KUKA KRL data list: CNC6.dat

&ACCESS RV
DEFDAT CNC6 Public
DECL GLOBAL FRAME gfCNCPoint6[13477]


gfCNCPoint6[1] = {X 105.3781, Y 13.7586, Z -8.0000, A 0.000, B 0.000, C 0.000 }
gfCNCPoint6[2] = {X 105.3083, Y 12.9780, Z -8.0000, A 0.000, B 0.000, C 0.000 }
gfCNCPoint6[3] = {X 105.3083, Y 12.1868, Z -8.0000, A 0.000, B 0.000, C 0.000 }
gfCNCPoint6[4] = {X 105.4186, Y 11.2077, Z -8.0000, A 0.000, B 0.000, C 0.000 }
gfCNCPoint6[5] = {X 105.7440, Y 10.2777, Z -8.0000, A 0.000, B 0.000, C 0.000 }
gfCNCPoint6[6] = {X 106.2682, Y 9.4435, Z -8.0000, A 0.000, B 0.000, C 0.000 }
gfCNCPoint6[7] = {X 106.9649, Y 8.7468, Z -8.0000, A 0.000, B 0.000, C 0.000 }
gfCNCPoint6[8] = {X 107.7992, Y 8.2226, Z -8.0000, A 0.000, B 0.000, C 0.000 }
gfCNCPoint6[9] = {X 108.7292, Y 7.8971, Z -8.0000, A 0.000, B 0.000, C 0.000 }
gfCNCPoint6[10] = {X 109.7083, Y 7.7868, Z -8.0000, A 0.000, B 0.000, C 0.000 }
gfCNCPoint6[11] = {X 117.7916, Y 7.7868, Z -8.0000, A 0.000, B 0.000, C 0.000 }
gfCNCPoint6[12] = {X 118.7707, Y 7.8971, Z -8.0000, A 0.000, B 0.000, C 0.000 }
gfCNCPoint6[13] = {X 119.7007, Y 8.2226, Z -8.0000, A 0.000, B 0.000, C 0.000 }
gfCNCPoint6[14] = {X 120.5349, Y 8.7468, Z -8.0000, A 0.000, B 0.000, C 0.000 }
gfCNCPoint6[15] = {X 121.2316, Y 9.4435, Z -8.0000, A 0.000, B 0.000, C 0.000 }
gfCNCPoint6[16] = {X 121.7558, Y 10.2777, Z -8.0000, A 0.000, B 0.000, C 0.000 }
gfCNCPoint6[17] = {X 122.0813, Y 11.2077, Z -8.0000, A 0.000, B 0.000, C 0.000 }
gfCNCPoint6[18] = {X 122.1916, Y 12.1868, Z -8.0000, A 0.000, B 0.000, C 0.000 }
gfCNCPoint6[19] = {X 122.1913, Y 13.0233, Z -8.0000, A 0.000, B 0.000, C 0.000 }
gfCNCPoint6[20] = {X 122.0831, Y 13.9490, Z -8.0000, A 0.000, B 0.000, C 0.000 }
gfCNCPoint6[21] = {X 121.7823, Y 14.8311, Z -8.0000, A 0.000, B 0.000, C 0.000 }
gfCNCPoint6[22] = {X 121.3025, Y 15.6301, Z -8.0000, A 0.000, B 0.000, C 0.000 }
gfCNCPoint6[23] = {X 120.6651, Y 16.3101, Z -8.0000, A 0.000, B 0.000, C 0.000 }
gfCNCPoint6[24] = {X 120.6653, Y 40.8772, Z -8.0000, A 0.000, B 0.000, C 0.000 }
gfCNCPoint6[25] = {X 120.6784, Y 40.8882, Z -8.0000, A 0.000, B 0.000, C 0.000 }
gfCNCPoint6[26] = {X 121.3172, Y 41.5763, Z -8.0000, A 0.000, B 0.000, C 0.000 }
gfCNCPoint6[27] = {X 121.7955, Y 42.3843, Z -8.0000, A 0.000, B 0.000, C 0.000 }
gfCNCPoint6[28] = {X 122.0914, Y 43.2753, Z -8.0000, A 0.000, B 0.000, C 0.000 }
gfCNCPoint6[29] = {X 122.1916, Y 44.2089, Z -8.0000, A 0.000, B 0.000, C 0.000 }
gfCNCPoint6[30] = {X 122.1916, Y 45.0000, Z -8.0000, A 0.000, B 0.000, C 0.000 }
gfCNCPoint6[31] = {X 122.0813, Y 45.9791, Z -8.0000, A 0.000, B 0.000, C 0.000 }
gfCNCPoint6[32] = {X 121.7558, Y 46.9091, Z -8.0000, A 0.000, B 0.000, C 0.000 }
gfCNCPoint6[33] = {X 121.2316, Y 47.7434, Z -8.0000, A 0.000, B 0.000, C 0.000 }
gfCNCPoint6[34] = {X 120.5349, Y 48.4401, Z -8.0000, A 0.000, B 0.000, C 0.000 }
gfCNCPoint6[35] = {X 119.7007, Y 48.9643, Z -8.0000, A 0.000, B 0.000, C 0.000 }
gfCNCPoint6[36] = {X 118.7707, Y 49.2897, Z -8.0000, A 0.000, B 0.000, C 0.000 }
gfCNCPoint6[37] = {X 117.7916, Y 49.4000, Z -8.0000, A 0.000, B 0.000, C 0.000 }
gfCNCPoint6[38] = {X 111.9185, Y 49.4000, Z -8.0000, A 0.000, B 0.000, C 0.000 }
gfCNCPoint6[39] = {X 110.9394, Y 49.2897, Z -8.0000, A 0.000, B 0.000, C 0.000 }
gfCNCPoint6[40] = {X 110.0094, Y 48.9643, Z -8.0000, A 0.000, B 0.000, C 0.000 }
gfCNCPoint6[41] = {X 109.1751, Y 48.4401, Z -8.0000, A 0.000, B 0.000, C 0.000 }
gfCNCPoint6[42] = {X 108.4784, Y 47.7433, Z -8.0000, A 0.000, B 0.000, C 0.000 }
gfCNCPoint6[43] = {X 107.9542, Y 46.9091, Z -8.0000, A 0.000, B 0.000, C 0.000 }
gfCNCPoint6[44] = {X 107.6288, Y 45.9791, Z -8.0000, A 0.000, B 0.000, C 0.000 }
gfCNCPoint6[45] = {X 107.5185, Y 45.0000, Z -8.0000, A 0.000, B 0.000, C 0.000 }
gfCNCPoint6[46] = {X 107.5185, Y 44.1753, Z -8.0000, A 0.000, B 0.000, C 0.000 }
gfCNCPoint6[47] = {X 107.5542, Y 43.6267, Z -8.0000, A 0.000, B 0.000, C 0.000 }
gfCNCPoint6[48] = {X 107.6609, Y 43.0873, Z -8.0000, A 0.000, B 0.000, C 0.000 }
gfCNCPoint6[49] = {X 106.1856, Y 46.6923, Z -8.0000, A 0.000, B 0.000, C 0.000 }
gfCNCPoint6[50] = {X 105.8087, Y 47.4049, Z -8.0000, A 0.000, B 0.000, C 0.000 }
gfCNCPoint6[51] = {X 105.3081, Y 48.0367, Z -8.0000, A 0.000, B 0.000, C 0.000 }
gfCNCPoint6[52] = {X 104.7006, Y 48.5667, Z -8.0000, A 0.000, B 0.000, C 0.000 }
gfCNCPoint6[53] = {X 104.0067, Y 48.9769, Z -8.0000, A 0.000, B 0.000, C 0.000 }
gfCNCPoint6[54] = {X 103.0414, Y 49.3033, Z -8.0000, A 0.000, B 0.000, C 0.000 }
gfCNCPoint6[55] = {X 102.0269, Y 49.3989, Z -8.0000, A 0.000, B 0.000, C 0.000 }
gfCNCPoint6[56] = {X 101.0176, Y 49.2586, Z -8.0000, A 0.000, B 0.000, C 0.000 }
gfCNCPoint6[57] = {X 100.0676, Y 48.8899, Z -8.0000, A 0.000, B 0.000, C 0.000 }
gfCNCPoint6[58] = {X 99.2280, Y 48.3125, Z -8.0000, A 0.000, B 0.000, C 0.000 }
gfCNCPoint6[59] = {X 98.5436, Y 47.5575, Z -8.0000, A 0.000, B 0.000, C 0.000 }
gfCNCPoint6[60] = {X 98.0514, Y 46.6653, Z -8.0000, A 0.000, B 0.000, C 0.000 }
gfCNCPoint6[61] = {X 96.5899, Y 43.0909, Z -8.0000, A 0.000, B 0.000, C 0.000 }
gfCNCPoint6[62] = {X 96.6995, Y 43.6452, Z -8.0000, A 0.000, B 0.000, C 0.000 }
gfCNCPoint6[63] = {X 96.7385, Y 44.2088, Z -8.0000, A 0.000, B 0.000, C 0.000 }
gfCNCPoint6[64] = {X 96.7383, Y 45.0423, Z -8.0000, A 0.000, B 0.000, C 0.000 }
gfCNCPoint6[65] = {X 96.6200, Y 46.0144, Z -8.0000, A 0.000, B 0.000, C 0.000 }
gfCNCPoint6[66] = {X 96.2896, Y 46.9363, Z -8.0000, A 0.000, B 0.000, C 0.000 }
gfCNCPoint6[67] = {X 95.7635, Y 47.7622, Z -8.0000, A 0.000, B 0.000, C 0.000 }
gfCNCPoint6[68] = {X 95.0677, Y 48.4513, Z -8.0000, A 0.000, B 0.000, C 0.000 }
gfCNCPoint6[69] = {X 94.2367, Y 48.9695, Z -8.0000, A 0.000, B 0.000, C 0.000 }
gfCNCPoint6[70] = {X 93.3117, Y 49.2910, Z -8.0000, A 0.000, B 0.000, C 0.000 }
gfCNCPoint6[71] = {X 92.3385, Y 49.4000, Z -8.0000, A 0.000, B 0.000, C 0.000 }
gfCNCPoint6[72] = {X 85.8951, Y 49.4000, Z -8.0000, A 0.000, B 0.000, C 0.000 }
gfCNCPoint6[73] = {X 84.9160, Y 49.2897, Z -8.0000, A 0.000, B 0.000, C 0.000 }
gfCNCPoint6[74] = {X 83.9860, Y 48.9643, Z -8.0000, A 0.000, B 0.000, C 0.000 }
gfCNCPoint6[75] = {X 83.1517, Y 48.4401, Z -8.0000, A 0.000, B 0.000, C 0.000 }
gfCNCPoint6[76] = {X 82.4550, Y 47.7433, Z -8.0000, A 0.000, B 0.000, C 0.000 }
gfCNCPoint6[77] = {X 81.9308, Y 46.9091, Z -8.0000, A 0.000, B 0.000, C 0.000 }
gfCNCPoint6[78] = {X 81.6054, Y 45.9791, Z -8.0000, A 0.000, B 0.000, C 0.000 }
gfCNCPoint6[79] = {X 81.4951, Y 45.0000, Z -8.0000, A 0.000, B 0.000, C 0.000 }
gfCNCPoint6[80] = {X 81.4951, Y 44.2069, Z -8.0000, A 0.000, B 0.000, C 0.000 }
gfCNCPoint6[81] = {X 81.5995, Y 43.2694, Z -8.0000, A 0.000, B 0.000, C 0.000 }
gfCNCPoint6[82] = {X 81.8990, Y 42.3749, Z -8.0000, A 0.000, B 0.000, C 0.000 }
gfCNCPoint6[83] = {X 82.3802, Y 41.5636, Z -8.0000, A 0.000, B 0.000, C 0.000 }
gfCNCPoint6[84] = {X 83.0216, Y 40.8719, Z -8.0000, A 0.000, B 0.000, C 0.000 }
gfCNCPoint6[85] = {X 83.0217, Y 16.3102, Z -8.0000, A 0.000, B 0.000, C 0.000 }
gfCNCPoint6[86] = {X 82.3774, Y 15.6212, Z -8.0000, A 0.000, B 0.000, C 0.000 }
gfCNCPoint6[87] = {X 81.8949, Y 14.8106, Z -8.0000, A 0.000, B 0.000, C 0.000 }
gfCNCPoint6[88] = {X 81.5962, Y 13.9159, Z -8.0000, A 0.000, B 0.000, C 0.000 }
gfCNCPoint6[89] = {X 81.4951, Y 12.9780, Z -8.0000, A 0.000, B 0.000, C 0.000 }
gfCNCPoint6[90] = {X 81.4951, Y 12.1868, Z -8.0000, A 0.000, B 0.000, C 0.000 }
gfCNCPoint6[91] = {X 81.5776, Y 11.3387, Z -8.0000, A 0.000, B 0.000, C 0.000 }
gfCNCPoint6[92] = {X 81.8220, Y 10.5225, Z -8.0000, A 0.000, B 0.000, C 0.000 }
gfCNCPoint6[93] = {X 82.2192, Y 9.7686, Z -8.0000, A 0.000, B 0.000, C 0.000 }
gfCNCPoint6[94] = {X 81.8181, Y 9.5048, Z -8.0000, A 0.000, B 0.000, C 0.000 }
gfCNCPoint6[95] = {X 68.9232, Y 9.5048, Z -8.0000, A 0.000, B 0.000, C 0.000 }
gfCNCPoint6[96] = {X 69.1905, Y 10.7207, Z -8.0000, A 0.000, B 0.000, C 0.000 }
gfCNCPoint6[97] = {X 69.2995, Y 11.9609, Z -8.0000, A 0.000, B 0.000, C 0.000 }
gfCNCPoint6[98] = {X 69.3015, Y 12.0738, Z -8.0000, A 0.000, B 0.000, C 0.000 }
gfCNCPoint6[99] = {X 69.3021, Y 12.1868, Z -8.0000, A 0.000, B 0.000, C 0.000 }
gfCNCPoint6[100] = {X 69.3017, Y 13.0686, Z -8.0000, A 0.000, B 0.000, C 0.000 }
gfCNCPoint6[101] = {X 69.2128, Y 14.2897, Z -8.0000, A 0.000, B 0.000, C 0.000 }
gfCNCPoint6[102] = {X 68.9706, Y 15.4898, Z -8.0000, A 0.000, B 0.000, C 0.000 }
gfCNCPoint6[103] = {X 76.9202, Y 36.7547, Z -8.0000, A 0.000, B 0.000, C 0.000 }
gfCNCPoint6[104] = {X 77.6316, Y 37.4066, Z -8.0000, A 0.000, B 0.000, C 0.000 }
gfCNCPoint6[105] = {X 78.2746, Y 38.1261, Z -8.0000, A 0.000, B 0.000, C 0.000 }
gfCNCPoint6[106] = {X 79.0225, Y 39.1911, Z -8.0000, A 0.000, B 0.000, C 0.000 }
gfCNCPoint6[107] = {X 79.6207, Y 40.3468, Z -8.0000, A 0.000, B 0.000, C 0.000 }
gfCNCPoint6[108] = {X 80.0585, Y 41.5723, Z -8.0000, A 0.000, B 0.000, C 0.000 }
gfCNCPoint6[109] = {X 80.3280, Y 42.8454, Z -8.0000, A 0.000, B 0.000, C 0.000 }
gfCNCPoint6[110] = {X 80.4242, Y 44.1432, Z -8.0000, A 0.000, B 0.000, C 0.000 }
gfCNCPoint6[111] = {X 80.4245, Y 45.0000, Z -8.0000, A 0.000, B 0.000, C 0.000 }
gfCNCPoint6[112] = {X 80.3511, Y 46.1898, Z -8.0000, A 0.000, B 0.000, C 0.000 }
gfCNCPoint6[113] = {X 80.1320, Y 47.3615, Z -8.0000, A 0.000, B 0.000, C 0.000 }
gfCNCPoint6[114] = {X 79.7706, Y 48.4974, Z -8.0000, A 0.000, B 0.000, C 0.000 }
gfCNCPoint6[115] = {X 79.2722, Y 49.5803, Z -8.0000, A 0.000, B 0.000, C 0.000 }
gfCNCPoint6[116] = {X 78.4688, Y 50.8341, Z -8.0000, A 0.000, B 0.000, C 0.000 }
gfCNCPoint6[117] = {X 77.4826, Y 51.9498, Z -8.0000, A 0.000, B 0.000, C 0.000 }
gfCNCPoint6[118] = {X 76.3369, Y 52.9011, Z -8.0000, A 0.000, B 0.000, C 0.000 }
gfCNCPoint6[119] = {X 75.0589, Y 53.6653, Z -8.0000, A 0.000, B 0.000, C 0.000 }
gfCNCPoint6[120] = {X 73.6787, Y 54.2246, Z -8.0000, A 0.000, B 0.000, C 0.000 }
gfCNCPoint6[121] = {X 72.2292, Y 54.5655, Z -8.0000, A 0.000, B 0.000, C 0.000 }
gfCNCPoint6[122] = {X 70.7445, Y 54.6800, Z -8.0000, A 0.000, B 0.000, C 0.000 }
gfCNCPoint6[123] = {X 64.1851, Y 54.6800, Z -8.0000, A 0.000, B 0.000, C 0.000 }
gfCNCPoint6[124] = {X 62.7229, Y 54.5689, Z -8.0000, A 0.000, B 0.000, C 0.000 }
gfCNCPoint6[125] = {X 61.2943, Y 54.2383, Z -8.0000, A 0.000, B 0.000, C 0.000 }
gfCNCPoint6[126] = {X 59.9320, Y 53.6956, Z -8.0000, A 0.000, B 0.000, C 0.000 }
gfCNCPoint6[127] = {X 58.6673, Y 52.9534, Z -8.0000, A 0.000, B 0.000, C 0.000 }
gfCNCPoint6[128] = {X 57.5293, Y 52.0286, Z -8.0000, A 0.000, B 0.000, C 0.000 }
gfCNCPoint6[129] = {X 56.6337, Y 51.0563, Z -8.0000, A 0.000, B 0.000, C 0.000 }
gfCNCPoint6[130] = {X 55.8790, Y 49.9710, Z -8.0000, A 0.000, B 0.000, C 0.000 }
gfCNCPoint6[131] = {X 55.1243, Y 51.0563, Z -8.0000, A 0.000, B 0.000, C 0.000 }
gfCNCPoint6[132] = {X 54.2288, Y 52.0286, Z -8.0000, A 0.000, B 0.000, C 0.000 }
gfCNCPoint6[133] = {X 53.0907, Y 52.9534, Z -8.0000, A 0.000, B 0.000, C 0.000 }
gfCNCPoint6[134] = {X 51.8261, Y 53.6956, Z -8.0000, A 0.000, B 0.000, C 0.000 }
gfCNCPoint6[135] = {X 50.4638, Y 54.2383, Z -8.0000, A 0.000, B 0.000, C 0.000 }
gfCNCPoint6[136] = {X 49.0351, Y 54.5689, Z -8.0000, A 0.000, B 0.000, C 0.000 }
gfCNCPoint6[137] = {X 47.5729, Y 54.6800, Z -8.0000, A 0.000, B 0.000, C 0.000 }
gfCNCPoint6[138] = {X 40.6393, Y 54.6800, Z -8.0000, A 0.000, B 0.000, C 0.000 }
gfCNCPoint6[139] = {X 39.2448, Y 54.5790, Z -8.0000, A 0.000, B 0.000, C 0.000 }
gfCNCPoint6[140] = {X 37.8793, Y 54.2782, Z -8.0000, A 0.000, B 0.000, C 0.000 }
gfCNCPoint6[141] = {X 36.5715, Y 53.7838, Z -8.0000, A 0.000, B 0.000, C 0.000 }
gfCNCPoint6[142] = {X 35.3485, Y 53.1062, Z -8.0000, A 0.000, B 0.000, C 0.000 }
gfCNCPoint6[143] = {X 33.9151, Y 54.1351, Z -8.0000, A 0.000, B 0.000, C 0.000 }
gfCNCPoint6[144] = {X 32.3637, Y 54.9757, Z -8.0000, A 0.000, B 0.000, C 0.000 }
gfCNCPoint6[145] = {X 30.7189, Y 55.6147, Z -8.0000, A 0.000, B 0.000, C 0.000 }
gfCNCPoint6[146] = {X 29.0069, Y 56.0418, Z -8.0000, A 0.000, B 0.000, C 0.000 }
gfCNCPoint6[147] = {X 27.2548, Y 56.2503, Z -8.0000, A 0.000, B 0.000, C 0.000 }
gfCNCPoint6[148] = {X 24.9805, Y 57.2333, Z -8.0000, A 0.000, B 0.000, C 0.000 }
gfCNCPoint6[149] = {X 22.6486, Y 58.0704, Z -8.0000, A 0.000, B 0.000, C 0.000 }
gfCNCPoint6[150] = {X 20.0864, Y 58.7995, Z -8.0000, A 0.000, B 0.000, C 0.000 }
gfCNCPoint6[151] = {X 17.4731, Y 59.3158, Z -8.0000, A 0.000, B 0.000, C 0.000 }
gfCNCPoint6[152] = {X 14.8262, Y 59.6160, Z -8.0000, A 0.000, B 0.000, C 0.000 }
gfCNCPoint6[153] = {X 12.1636, Y 59.6979, Z -8.0000, A 0.000, B 0.000, C 0.000 }
gfCNCPoint6[154] = {X 9.5033, Y 59.5611, Z -8.0000, A 0.000, B 0.000, C 0.000 }
gfCNCPoint6[155] = {X 9.5033, Y 90.4952, Z -8.0000, A 0.000, B 0.000, C 0.000 }
gfCNCPoint6[156] = {X 114.8634, Y 90.4952, Z -8.0000, A 0.000, B 0.000, C 0.000 }
gfCNCPoint6[157] = {X 115.7474, Y 89.2996, Z -8.0000, A 0.000, B 0.000, C 0.000 }
gfCNCPoint6[158] = {X 116.7717, Y 88.2217, Z -8.0000, A 0.000, B 0.000, C 0.000 }
gfCNCPoint6[159] = {X 117.9206, Y 87.2778, Z -8.0000, A 0.000, B 0.000, C 0.000 }
gfCNCPoint6[160] = {X 119.1768, Y 86.4822, Z -8.0000, A 0.000, B 0.000, C 0.000 }
gfCNCPoint6[161] = {X 120.5212, Y 85.8469, Z -8.0000, A 0.000, B 0.000, C 0.000 }
gfCNCPoint6[162] = {X 121.9334, Y 85.3816, Z -8.0000, A 0.000, B 0.000, C 0.000 }
gfCNCPoint6[163] = {X 123.3922, Y 85.0934, Z -8.0000, A 0.000, B 0.000, C 0.000 }
gfCNCPoint6[164] = {X 123.5272, Y 84.9476, Z -8.0000, A 0.000, B 0.000, C 0.000 }
gfCNCPoint6[165] = {X 123.6609, Y 84.8006, Z -8.0000, A 0.000, B 0.000, C 0.000 }
gfCNCPoint6[166] = {X 147.2181, Y 58.9332, Z -8.0000, A 0.000, B 0.000, C 0.000 }
gfCNCPoint6[167] = {X 147.2180, Y 58.0000, Z -8.0000, A 0.000, B 0.000, C 0.000 }
gfCNCPoint6[168] = {X 147.2987, Y 56.6058, Z -8.0000, A 0.000, B 0.000, C 0.000 }
gfCNCPoint6[169] = {X 147.5398, Y 55.2303, Z -8.0000, A 0.000, B 0.000, C 0.000 }
gfCNCPoint6[170] = {X 148.0022, Y 53.7185, Z -8.0000, A 0.000, B 0.000, C 0.000 }
gfCNCPoint6[171] = {X 148.6580, Y 52.2800, Z -8.0000, A 0.000, B 0.000, C 0.000 }
gfCNCPoint6[172] = {X 143.0396, Y 52.2800, Z -8.0000, A 0.000, B 0.000, C 0.000 }
gfCNCPoint6[173] = {X 141.7807, Y 52.1703, Z -8.0000, A 0.000, B 0.000, C 0.000 }
gfCNCPoint6[174] = {X 140.5597, Y 51.8446, Z -8.0000, A 0.000, B 0.000, C 0.000 }
gfCNCPoint6[175] = {X 139.4134, Y 51.3126, Z -8.0000, A 0.000, B 0.000, C 0.000 }
gfCNCPoint6[176] = {X 138.3764, Y 50.5904, Z -8.0000, A 0.000, B 0.000, C 0.000 }
gfCNCPoint6[177] = {X 137.4799, Y 49.6998, Z -8.0000, A 0.000, B 0.000, C 0.000 }
gfCNCPoint6[178] = {X 136.7509, Y 48.6675, Z -8.0000, A 0.000, B 0.000, C 0.000 }
gfCNCPoint6[179] = {X 136.2114, Y 47.5248, Z -8.0000, A 0.000, B 0.000, C 0.000 }
gfCNCPoint6[180] = {X 135.8777, Y 46.3059, Z -8.0000, A 0.000, B 0.000, C 0.000 }
gfCNCPoint6[181] = {X 135.7598, Y 45.0477, Z -8.0000, A 0.000, B 0.000, C 0.000 }
gfCNCPoint6[182] = {X 135.7601, Y 44.1248, Z -8.0000, A 0.000, B 0.000, C 0.000 }
gfCNCPoint6[183] = {X 135.8408, Y 43.1249, Z -8.0000, A 0.000, B 0.000, C 0.000 }
gfCNCPoint6[184] = {X 136.0581, Y 42.1457, Z -8.0000, A 0.000, B 0.000, C 0.000 }
gfCNCPoint6[185] = {X 138.3597, Y 42.8258, Z -8.0000, A 0.000, B 0.000, C 0.000 }
gfCNCPoint6[186] = {X 138.6721, Y 42.0319, Z -8.0000, A 0.000, B 0.000, C 0.000 }
gfCNCPoint6[187] = {X 139.1179, Y 41.3046, Z -8.0000, A 0.000, B 0.000, C 0.000 }
gfCNCPoint6[188] = {X 139.6836, Y 40.6660, Z -8.0000, A 0.000, B 0.000, C 0.000 }
gfCNCPoint6[189] = {X 139.6836, Y 20.4384, Z -8.0000, A 0.000, B 0.000, C 0.000 }
gfCNCPoint6[190] = {X 137.7093, Y 20.4382, Z -8.0000, A 0.000, B 0.000, C 0.000 }
gfCNCPoint6[191] = {X 136.9994, Y 21.1828, Z -8.0000, A 0.000, B 0.000, C 0.000 }
gfCNCPoint6[192] = {X 136.1491, Y 21.7619, Z -8.0000, A 0.000, B 0.000, C 0.000 }
gfCNCPoint6[193] = {X 135.4282, Y 22.0767, Z -8.0000, A 0.000, B 0.000, C 0.000 }
gfCNCPoint6[194] = {X 134.6660, Y 22.2715, Z -8.0000, A 0.000, B 0.000, C 0.000 }
gfCNCPoint6[195] = {X 133.8824, Y 22.3414, Z -8.0000, A 0.000, B 0.000, C 0.000 }
gfCNCPoint6[196] = {X 133.2006, Y 22.3415, Z -8.0000, A 0.000, B 0.000, C 0.000 }
gfCNCPoint6[197] = {X 132.2486, Y 22.2478, Z -8.0000, A 0.000, B 0.000, C 0.000 }
gfCNCPoint6[198] = {X 131.3331, Y 21.9701, Z -8.0000, A 0.000, B 0.000, C 0.000 }
gfCNCPoint6[199] = {X 130.4895, Y 21.5191, Z -8.0000, A 0.000, B 0.000, C 0.000 }
gfCNCPoint6[200] = {X 129.7500, Y 20.9122, Z -8.0000, A 0.000, B 0.000, C 0.000 }
gfCNCPoint6[201] = {X 129.1431, Y 20.1727, Z -8.0000, A 0.000, B 0.000, C 0.000 }
gfCNCPoint6[202] = {X 128.6921, Y 19.3290, Z -8.0000, A 0.000, B 0.000, C 0.000 }
gfCNCPoint6[203] = {X 128.4144, Y 18.4136, Z -8.0000, A 0.000, B 0.000, C 0.000 }
gfCNCPoint6[204] = {X 128.3206, Y 17.4615, Z -8.0000, A 0.000, B 0.000, C 0.000 }
gfCNCPoint6[205] = {X 128.3206, Y 10.4835, Z -8.0000, A 0.000, B 0.000, C 0.000 }
gfCNCPoint6[206] = {X 128.3317, Y 10.1547, Z -8.0000, A 0.000, B 0.000, C 0.000 }
gfCNCPoint6[207] = {X 128.3649, Y 9.8275, Z -8.0000, A 0.000, B 0.000, C 0.000 }
gfCNCPoint6[208] = {X 128.6079, Y 8.8340, Z -8.0000, A 0.000, B 0.000, C 0.000 }
gfCNCPoint6[209] = {X 129.0526, Y 7.9130, Z -8.0000, A 0.000, B 0.000, C 0.000 }
gfCNCPoint6[210] = {X 129.6794, Y 7.1048, Z -8.0000, A 0.000, B 0.000, C 0.000 }
gfCNCPoint6[211] = {X 130.0258, Y 7.4372, Z -8.0000, A 0.000, B 0.000, C 0.000 }
gfCNCPoint6[212] = {X 130.6998, Y 6.8633, Z -8.0000, A 0.000, B 0.000, C 0.000 }
gfCNCPoint6[213] = {X 131.4750, Y 6.4360, Z -8.0000, A 0.000, B 0.000, C 0.000 }
gfCNCPoint6[214] = {X 132.3200, Y 6.1725, Z -8.0000, A 0.000, B 0.000, C 0.000 }
gfCNCPoint6[215] = {X 133.2007, Y 6.0835, Z -8.0000, A 0.000, B 0.000, C 0.000 }
gfCNCPoint6[216] = {X 133.8874, Y 6.0837, Z -8.0000, A 0.000, B 0.000, C 0.000 }
gfCNCPoint6[217] = {X 134.7185, Y 6.1716, Z -8.0000, A 0.000, B 0.000, C 0.000 }
gfCNCPoint6[218] = {X 135.5180, Y 6.4151, Z -8.0000, A 0.000, B 0.000, C 0.000 }
gfCNCPoint6[219] = {X 136.2570, Y 6.8053, Z -8.0000, A 0.000, B 0.000, C 0.000 }
gfCNCPoint6[220] = {X 136.9090, Y 7.3283, Z -8.0000, A 0.000, B 0.000, C 0.000 }
gfCNCPoint6[221] = {X 137.4502, Y 7.9650, Z -8.0000, A 0.000, B 0.000, C 0.000 }
gfCNCPoint6[222] = {X 155.0725, Y 7.9650, Z -8.0000, A 0.000, B 0.000, C 0.000 }
gfCNCPoint6[223] = {X 155.6203, Y 7.3220, Z -8.0000, A 0.000, B 0.000, C 0.000 }
gfCNCPoint6[224] = {X 156.2808, Y 6.7954, Z -8.0000, A 0.000, B 0.000, C 0.000 }
gfCNCPoint6[225] = {X 157.0298, Y 6.4048, Z -8.0000, A 0.000, B 0.000, C 0.000 }
gfCNCPoint6[226] = {X 157.8397, Y 6.1646, Z -8.0000, A 0.000, B 0.000, C 0.000 }
gfCNCPoint6[227] = {X 158.6805, Y 6.0835, Z -8.0000, A 0.000, B 0.000, C 0.000 }
gfCNCPoint6[228] = {X 159.3791, Y 6.0839, Z -8.0000, A 0.000, B 0.000, C 0.000 }
gfCNCPoint6[229] = {X 160.3488, Y 6.2050, Z -8.0000, A 0.000, B 0.000, C 0.000 }
gfCNCPoint6[230] = {X 161.2678, Y 6.5371, Z -8.0000, A 0.000, B 0.000, C 0.000 }
gfCNCPoint6[231] = {X 162.0908, Y 7.0639, Z -8.0000, A 0.000, B 0.000, C 0.000 }
gfCNCPoint6[232] = {X 162.7773, Y 7.7593, Z -8.0000, A 0.000, B 0.000, C 0.000 }
gfCNCPoint6[233] = {X 163.2934, Y 8.5891, Z -8.0000, A 0.000, B 0.000, C 0.000 }
gfCNCPoint6[234] = {X 163.6136, Y 9.5124, Z -8.0000, A 0.000, B 0.000, C 0.000 }
gfCNCPoint6[235] = {X 163.7221, Y 10.4835, Z -8.0000, A 0.000, B 0.000, C 0.000 }
gfCNCPoint6[236] = {X 163.7221, Y 17.4615, Z -8.0000, A 0.000, B 0.000, C 0.000 }
gfCNCPoint6[237] = {X 163.6118, Y 18.4406, Z -8.0000, A 0.000, B 0.000, C 0.000 }
gfCNCPoint6[238] = {X 163.2863, Y 19.3706, Z -8.0000, A 0.000, B 0.000, C 0.000 }
gfCNCPoint6[239] = {X 162.7621, Y 20.2049, Z -8.0000, A 0.000, B 0.000, C 0.000 }
gfCNCPoint6[240] = {X 162.0654, Y 20.9016, Z -8.0000, A 0.000, B 0.000, C 0.000 }
gfCNCPoint6[241] = {X 161.2312, Y 21.4258, Z -8.0000, A 0.000, B 0.000, C 0.000 }
gfCNCPoint6[242] = {X 160.3012, Y 21.7512, Z -8.0000, A 0.000, B 0.000, C 0.000 }
gfCNCPoint6[243] = {X 159.3221, Y 21.8615, Z -8.0000, A 0.000, B 0.000, C 0.000 }
gfCNCPoint6[244] = {X 158.6792, Y 21.8615, Z -8.0000, A 0.000, B 0.000, C 0.000 }
gfCNCPoint6[245] = {X 157.8337, Y 21.7773, Z -8.0000, A 0.000, B 0.000, C 0.000 }
gfCNCPoint6[246] = {X 157.0198, Y 21.5332, Z -8.0000, A 0.000, B 0.000, C 0.000 }
gfCNCPoint6[247] = {X 156.2675, Y 21.1381, Z -8.0000, A 0.000, B 0.000, C 0.000 }
gfCNCPoint6[248] = {X 155.6045, Y 20.6066, Z -8.0000, A 0.000, B 0.000, C 0.000 }
gfCNCPoint6[249] = {X 155.0552, Y 19.9583, Z -8.0000, A 0.000, B 0.000, C 0.000 }
gfCNCPoint6[250] = {X 152.3574, Y 19.9591, Z -8.0000, A 0.000, B 0.000, C 0.000 }
gfCNCPoint6[251] = {X 152.3564, Y 40.8428, Z -8.0000, A 0.000, B 0.000, C 0.000 }
gfCNCPoint6[252] = {X 152.8071, Y 41.3287, Z -8.0000, A 0.000, B 0.000, C 0.000 }
gfCNCPoint6[253] = {X 152.9013, Y 41.4409, Z -8.0000, A 0.000, B 0.000, C 0.000 }
gfCNCPoint6[254] = {X 153.4357, Y 42.2811, Z -8.0000, A 0.000, B 0.000, C 0.000 }
gfCNCPoint6[255] = {X 153.7686, Y 43.2196, Z -8.0000, A 0.000, B 0.000, C 0.000 }
gfCNCPoint6[256] = {X 153.8831, Y 44.2088, Z -8.0000, A 0.000, B 0.000, C 0.000 }
gfCNCPoint6[257] = {X 153.8829, Y 45.0423, Z -8.0000, A 0.000, B 0.000, C 0.000 }
gfCNCPoint6[258] = {X 153.7646, Y 46.0144, Z -8.0000, A 0.000, B 0.000, C 0.000 }
gfCNCPoint6[259] = {X 153.4342, Y 46.9363, Z -8.0000, A 0.000, B 0.000, C 0.000 }
gfCNCPoint6[260] = {X 152.9080, Y 47.7622, Z -8.0000, A 0.000, B 0.000, C 0.000 }
gfCNCPoint6[261] = {X 152.2123, Y 48.4513, Z -8.0000, A 0.000, B 0.000, C 0.000 }
gfCNCPoint6[262] = {X 151.3813, Y 48.9695, Z -8.0000, A 0.000, B 0.000, C 0.000 }
gfCNCPoint6[263] = {X 150.4563, Y 49.2910, Z -8.0000, A 0.000, B 0.000, C 0.000 }
gfCNCPoint6[264] = {X 149.4831, Y 49.4000, Z -8.0000, A 0.000, B 0.000, C 0.000 }
gfCNCPoint6[265] = {X 143.0396, Y 49.4000, Z -8.0000, A 0.000, B 0.000, C 0.000 }
gfCNCPoint6[266] = {X 142.0605, Y 49.2897, Z -8.0000, A 0.000, B 0.000, C 0.000 }
gfCNCPoint6[267] = {X 141.1305, Y 48.9643, Z -8.0000, A 0.000, B 0.000, C 0.000 }
gfCNCPoint6[268] = {X 140.2963, Y 48.4401, Z -8.0000, A 0.000, B 0.000, C 0.000 }
gfCNCPoint6[269] = {X 139.5996, Y 47.7433, Z -8.0000, A 0.000, B 0.000, C 0.000 }
gfCNCPoint6[270] = {X 139.0754, Y 46.9091, Z -8.0000, A 0.000, B 0.000, C 0.000 }
gfCNCPoint6[271] = {X 138.7499, Y 45.9791, Z -8.0000, A 0.000, B 0.000, C 0.000 }
gfCNCPoint6[272] = {X 138.6396, Y 45.0000, Z -8.0000, A 0.000, B 0.000, C 0.000 }
gfCNCPoint6[273] = {X 138.6400, Y 44.1483, Z -8.0000, A 0.000, B 0.000, C 0.000 }
gfCNCPoint6[274] = {X 138.7505, Y 43.2275, Z -8.0000, A 0.000, B 0.000, C 0.000 }
gfCNCPoint6[275] = {X 139.0514, Y 42.3503, Z -8.0000, A 0.000, B 0.000, C 0.000 }
gfCNCPoint6[276] = {X 139.5295, Y 41.5556, Z -8.0000, A 0.000, B 0.000, C 0.000 }
gfCNCPoint6[277] = {X 140.1636, Y 40.8789, Z -8.0000, A 0.000, B 0.000, C 0.000 }
gfCNCPoint6[278] = {X 140.1636, Y 19.9585, Z -8.0000, A 0.000, B 0.000, C 0.000 }
gfCNCPoint6[279] = {X 137.4654, Y 19.9582, Z -8.0000, A 0.000, B 0.000, C 0.000 }
gfCNCPoint6[280] = {X 136.9177, Y 20.6083, Z -8.0000, A 0.000, B 0.000, C 0.000 }
gfCNCPoint6[281] = {X 136.2552, Y 21.1409, Z -8.0000, A 0.000, B 0.000, C 0.000 }
gfCNCPoint6[282] = {X 135.5027, Y 21.5362, Z -8.0000, A 0.000, B 0.000, C 0.000 }
gfCNCPoint6[283] = {X 134.6883, Y 21.7794, Z -8.0000, A 0.000, B 0.000, C 0.000 }
gfCNCPoint6[284] = {X 133.8422, Y 21.8615, Z -8.0000, A 0.000, B 0.000, C 0.000 }
gfCNCPoint6[285] = {X 133.2006, Y 21.8615, Z -8.0000, A 0.000, B 0.000, C 0.000 }
gfCNCPoint6[286] = {X 132.2215, Y 21.7512, Z -8.0000, A 0.000, B 0.000, C 0.000 }
gfCNCPoint6[287] = {X 131.2916, Y 21.4258, Z -8.0000, A 0.000, B 0.000, C 0.000 }
gfCNCPoint6[288] = {X 130.4573, Y 20.9016, Z -8.0000, A 0.000, B 0.000, C 0.000 }
gfCNCPoint6[289] = {X 129.7606, Y 20.2049, Z -8.0000, A 0.000, B 0.000, C 0.000 }
gfCNCPoint6[290] = {X 129.2364, Y 19.3706, Z -8.0000, A 0.000, B 0.000, C 0.000 }
gfCNCPoint6[291] = {X 128.9110, Y 18.4406, Z -8.0000, A 0.000, B 0.000, C 0.000 }
gfCNCPoint6[292] = {X 128.8006, Y 17.4615, Z -8.0000, A 0.000, B 0.000, C 0.000 }
gfCNCPoint6[293] = {X 128.8006, Y 10.4835, Z -8.0000, A 0.000, B 0.000, C 0.000 }
gfCNCPoint6[294] = {X 128.8808, Y 9.6474, Z -8.0000, A 0.000, B 0.000, C 0.000 }
gfCNCPoint6[295] = {X 129.1184, Y 8.8418, Z -8.0000, A 0.000, B 0.000, C 0.000 }
gfCNCPoint6[296] = {X 129.5048, Y 8.0960, Z -8.0000, A 0.000, B 0.000, C 0.000 }
gfCNCPoint6[297] = {X 130.0258, Y 7.4372, Z -8.0000, A 0.000, B 0.000, C 0.000 }
gfCNCPoint6[298] = {X 129.6794, Y 7.1048, Z -8.0000, A 0.000, B 0.000, C 0.000 }
gfCNCPoint6[299] = {X 102.4337, Y 7.1048, Z -8.0000, A 0.000, B 0.000, C 0.000 }
gfCNCPoint6[300] = {X 102.4337, Y 11.9048, Z -8.0000, A 0.000, B 0.000, C 0.000 }
gfCNCPoint6[301] = {X 101.3242, Y 11.9048, Z -8.0000, A 0.000, B 0.000, C 0.000 }
gfCNCPoint6[302] = {X 101.3283, Y 12.0458, Z -8.0000, A 0.000, B 0.000, C 0.000 }
gfCNCPoint6[303] = {X 101.3297, Y 12.1868, Z -8.0000, A 0.000, B 0.000, C 0.000 }
gfCNCPoint6[304] = {X 101.3293, Y 13.0462, Z -8.0000, A 0.000, B 0.000, C 0.000 }
gfCNCPoint6[305] = {X 101.2276, Y 14.1928, Z -8.0000, A 0.000, B 0.000, C 0.000 }
gfCNCPoint6[306] = {X 100.9464, Y 15.3090, Z -8.0000, A 0.000, B 0.000, C 0.000 }
gfCNCPoint6[307] = {X 101.3187, Y 16.2359, Z -8.0000, A 0.000, B 0.000, C 0.000 }
gfCNCPoint6[308] = {X 101.8679, Y 17.5961, Z -8.0000, A 0.000, B 0.000, C 0.000 }
gfCNCPoint6[309] = {X 102.6897, Y 15.5479, Z -8.0000, A 0.000, B 0.000, C 0.000 }
gfCNCPoint6[310] = {X 102.7997, Y 15.2735, Z -8.0000, A 0.000, B 0.000, C 0.000 }
gfCNCPoint6[311] = {X 102.5272, Y 14.1739, Z -8.0000, A 0.000, B 0.000, C 0.000 }
gfCNCPoint6[312] = {X 102.4286, Y 13.0454, Z -8.0000, A 0.000, B 0.000, C 0.000 }
gfCNCPoint6[313] = {X 102.4283, Y 12.1868, Z -8.0000, A 0.000, B 0.000, C 0.000 }
gfCNCPoint6[314] = {X 102.4296, Y 12.0458, Z -8.0000, A 0.000, B 0.000, C 0.000 }
gfCNCPoint6[315] = {X 102.4337, Y 11.9048, Z -8.0000, A 0.000, B 0.000, C 0.000 }
gfCNCPoint6[316] = {X 102.4337, Y 9.5048, Z -8.0000, A 0.000, B 0.000, C 0.000 }
gfCNCPoint6[317] = {X 98.1266, Y 9.5048, Z -8.0000, A 0.000, B 0.000, C 0.000 }
gfCNCPoint6[318] = {X 98.5429, Y 10.2827, Z -8.0000, A 0.000, B 0.000, C 0.000 }
gfCNCPoint6[319] = {X 98.8123, Y 11.1229, Z -8.0000, A 0.000, B 0.000, C 0.000 }
gfCNCPoint6[320] = {X 98.9260, Y 11.9978, Z -8.0000, A 0.000, B 0.000, C 0.000 }
gfCNCPoint6[321] = {X 98.9288, Y 12.0923, Z -8.0000, A 0.000, B 0.000, C 0.000 }
gfCNCPoint6[322] = {X 98.9297, Y 12.1868, Z -8.0000, A 0.000, B 0.000, C 0.000 }
gfCNCPoint6[323] = {X 98.9294, Y 13.0237, Z -8.0000, A 0.000, B 0.000, C 0.000 }
gfCNCPoint6[324] = {X 98.8590, Y 13.8052, Z -8.0000, A 0.000, B 0.000, C 0.000 }
gfCNCPoint6[325] = {X 98.6643, Y 14.5654, Z -8.0000, A 0.000, B 0.000, C 0.000 }
gfCNCPoint6[326] = {X 98.3502, Y 15.2845, Z -8.0000, A 0.000, B 0.000, C 0.000 }
gfCNCPoint6[327] = {X 99.0924, Y 17.1324, Z -8.0000, A 0.000, B 0.000, C 0.000 }
gfCNCPoint6[328] = {X 101.8751, Y 24.0238, Z -8.0000, A 0.000, B 0.000, C 0.000 }
gfCNCPoint6[329] = {X 104.9172, Y 16.4412, Z -8.0000, A 0.000, B 0.000, C 0.000 }
gfCNCPoint6[330] = {X 105.3924, Y 15.2557, Z -8.0000, A 0.000, B 0.000, C 0.000 }
gfCNCPoint6[331] = {X 105.0866, Y 14.5446, Z -8.0000, A 0.000, B 0.000, C 0.000 }
gfCNCPoint6[332] = {X 104.8970, Y 13.7941, Z -8.0000, A 0.000, B 0.000, C 0.000 }
gfCNCPoint6[333] = {X 104.8285, Y 13.0231, Z -8.0000, A 0.000, B 0.000, C 0.000 }
gfCNCPoint6[334] = {X 104.8283, Y 12.1868, Z -8.0000, A 0.000, B 0.000, C 0.000 }
gfCNCPoint6[335] = {X 104.8292, Y 12.0923, Z -8.0000, A 0.000, B 0.000, C 0.000 }
gfCNCPoint6[336] = {X 104.8319, Y 11.9978, Z -8.0000, A 0.000, B 0.000, C 0.000 }
gfCNCPoint6[337] = {X 104.9457, Y 11.1229, Z -8.0000, A 0.000, B 0.000, C 0.000 }
gfCNCPoint6[338] = {X 105.2151, Y 10.2827, Z -8.0000, A 0.000, B 0.000, C 0.000 }
gfCNCPoint6[339] = {X 105.6313, Y 9.5048, Z -8.0000, A 0.000, B 0.000, C 0.000 }
gfCNCPoint6[340] = {X 102.4337, Y 9.5048, Z -8.0000, A 0.000, B 0.000, C 0.000 }
gfCNCPoint6[341] = {X 102.4337, Y 7.1048, Z -8.0000, A 0.000, B 0.000, C 0.000 }
gfCNCPoint6[342] = {X 64.8348, Y 7.1048, Z -8.0000, A 0.000, B 0.000, C 0.000 }
gfCNCPoint6[343] = {X 65.5945, Y 8.0240, Z -8.0000, A 0.000, B 0.000, C 0.000 }
gfCNCPoint6[344] = {X 66.1940, Y 9.0549, Z -8.0000, A 0.000, B 0.000, C 0.000 }
gfCNCPoint6[345] = {X 66.6171, Y 10.1698, Z -8.0000, A 0.000, B 0.000, C 0.000 }
gfCNCPoint6[346] = {X 66.8305, Y 11.1683, Z -8.0000, A 0.000, B 0.000, C 0.000 }
gfCNCPoint6[347] = {X 66.9021, Y 12.1868, Z -8.0000, A 0.000, B 0.000, C 0.000 }
gfCNCPoint6[348] = {X 66.9018, Y 13.0462, Z -8.0000, A 0.000, B 0.000, C 0.000 }
gfCNCPoint6[349] = {X 66.7774, Y 14.3201, Z -8.0000, A 0.000, B 0.000, C 0.000 }
gfCNCPoint6[350] = {X 66.4317, Y 15.5524, Z -8.0000, A 0.000, B 0.000, C 0.000 }
gfCNCPoint6[351] = {X 74.9135, Y 38.2407, Z -8.0000, A 0.000, B 0.000, C 0.000 }
gfCNCPoint6[352] = {X 75.8052, Y 38.9755, Z -8.0000, A 0.000, B 0.000, C 0.000 }
gfCNCPoint6[353] = {X 76.5695, Y 39.8422, Z -8.0000, A 0.000, B 0.000, C 0.000 }
gfCNCPoint6[354] = {X 77.1870, Y 40.8188, Z -8.0000, A 0.000, B 0.000, C 0.000 }
gfCNCPoint6[355] = {X 77.6422, Y 41.8809, Z -8.0000, A 0.000, B 0.000, C 0.000 }
gfCNCPoint6[356] = {X 77.9237, Y 43.0016, Z -8.0000, A 0.000, B 0.000, C 0.000 }
gfCNCPoint6[357] = {X 78.0243, Y 44.1527, Z -8.0000, A 0.000, B 0.000, C 0.000 }
gfCNCPoint6[358] = {X 78.0245, Y 45.0000, Z -8.0000, A 0.000, B 0.000, C 0.000 }
gfCNCPoint6[359] = {X 77.9139, Y 46.2642, Z -8.0000, A 0.000, B 0.000, C 0.000 }
gfCNCPoint6[360] = {X 77.5854, Y 47.4899, Z -8.0000, A 0.000, B 0.000, C 0.000 }
gfCNCPoint6[361] = {X 77.0491, Y 48.6400, Z -8.0000, A 0.000, B 0.000, C 0.000 }
gfCNCPoint6[362] = {X 76.3213, Y 49.6795, Z -8.0000, A 0.000, B 0.000, C 0.000 }
gfCNCPoint6[363] = {X 75.4240, Y 50.5768, Z -8.0000, A 0.000, B 0.000, C 0.000 }
gfCNCPoint6[364] = {X 74.3845, Y 51.3047, Z -8.0000, A 0.000, B 0.000, C 0.000 }
gfCNCPoint6[365] = {X 73.2344, Y 51.8410, Z -8.0000, A 0.000, B 0.000, C 0.000 }
gfCNCPoint6[366] = {X 72.0086, Y 52.1694, Z -8.0000, A 0.000, B 0.000, C 0.000 }
gfCNCPoint6[367] = {X 70.7445, Y 52.2800, Z -8.0000, A 0.000, B 0.000, C 0.000 }
gfCNCPoint6[368] = {X 64.1851, Y 52.2800, Z -8.0000, A 0.000, B 0.000, C 0.000 }
gfCNCPoint6[369] = {X 62.9397, Y 52.1727, Z -8.0000, A 0.000, B 0.000, C 0.000 }
gfCNCPoint6[370] = {X 61.7311, Y 51.8539, Z -8.0000, A 0.000, B 0.000, C 0.000 }
gfCNCPoint6[371] = {X 60.5947, Y 51.3330, Z -8.0000, A 0.000, B 0.000, C 0.000 }
gfCNCPoint6[372] = {X 59.5643, Y 50.6255, Z -8.0000, A 0.000, B 0.000, C 0.000 }
gfCNCPoint6[373] = {X 58.6700, Y 49.7521, Z -8.0000, A 0.000, B 0.000, C 0.000 }
gfCNCPoint6[374] = {X 57.9384, Y 48.7385, Z -8.0000, A 0.000, B 0.000, C 0.000 }
gfCNCPoint6[375] = {X 57.3706, Y 47.5614, Z -8.0000, A 0.000, B 0.000, C 0.000 }
gfCNCPoint6[376] = {X 57.0224, Y 46.3017, Z -8.0000, A 0.000, B 0.000, C 0.000 }
gfCNCPoint6[377] = {X 56.9051, Y 45.0000, Z -8.0000, A 0.000, B 0.000, C 0.000 }
gfCNCPoint6[378] = {X 56.9052, Y 44.1968, Z -8.0000, A 0.000, B 0.000, C 0.000 }
gfCNCPoint6[379] = {X 56.9289, Y 43.6212, Z -8.0000, A 0.000, B 0.000, C 0.000 }
gfCNCPoint6[380] = {X 56.9981, Y 43.0492, Z -8.0000, A 0.000, B 0.000, C 0.000 }
gfCNCPoint6[381] = {X 54.7600, Y 43.0492, Z -8.0000, A 0.000, B 0.000, C 0.000 }
gfCNCPoint6[382] = {X 54.8275, Y 43.6012, Z -8.0000, A 0.000, B 0.000, C 0.000 }
gfCNCPoint6[383] = {X 54.8528, Y 44.1567, Z -8.0000, A 0.000, B 0.000, C 0.000 }
gfCNCPoint6[384] = {X 54.8529, Y 45.0000, Z -8.0000, A 0.000, B 0.000, C 0.000 }
gfCNCPoint6[385] = {X 54.7356, Y 46.3017, Z -8.0000, A 0.000, B 0.000, C 0.000 }
gfCNCPoint6[386] = {X 54.3875, Y 47.5614, Z -8.0000, A 0.000, B 0.000, C 0.000 }
gfCNCPoint6[387] = {X 53.8197, Y 48.7385, Z -8.0000, A 0.000, B 0.000, C 0.000 }
gfCNCPoint6[388] = {X 53.0880, Y 49.7521, Z -8.0000, A 0.000, B 0.000, C 0.000 }
gfCNCPoint6[389] = {X 52.1938, Y 50.6255, Z -8.0000, A 0.000, B 0.000, C 0.000 }
gfCNCPoint6[390] = {X 51.1633, Y 51.3330, Z -8.0000, A 0.000, B 0.000, C 0.000 }
gfCNCPoint6[391] = {X 50.0270, Y 51.8539, Z -8.0000, A 0.000, B 0.000, C 0.000 }
gfCNCPoint6[392] = {X 48.8183, Y 52.1727, Z -8.0000, A 0.000, B 0.000, C 0.000 }
gfCNCPoint6[393] = {X 47.5729, Y 52.2800, Z -8.0000, A 0.000, B 0.000, C 0.000 }
gfCNCPoint6[394] = {X 40.6393, Y 52.2800, Z -8.0000, A 0.000, B 0.000, C 0.000 }
gfCNCPoint6[395] = {X 39.4476, Y 52.1818, Z -8.0000, A 0.000, B 0.000, C 0.000 }
gfCNCPoint6[396] = {X 38.2881, Y 51.8899, Z -8.0000, A 0.000, B 0.000, C 0.000 }
gfCNCPoint6[397] = {X 37.1919, Y 51.4120, Z -8.0000, A 0.000, B 0.000, C 0.000 }
gfCNCPoint6[398] = {X 36.1888, Y 50.7612, Z -8.0000, A 0.000, B 0.000, C 0.000 }
gfCNCPoint6[399] = {X 35.3058, Y 49.9550, Z -8.0000, A 0.000, B 0.000, C 0.000 }
gfCNCPoint6[400] = {X 34.8234, Y 50.4196, Z -8.0000, A 0.000, B 0.000, C 0.000 }
gfCNCPoint6[401] = {X 34.3150, Y 50.8555, Z -8.0000, A 0.000, B 0.000, C 0.000 }
gfCNCPoint6[402] = {X 33.7814, Y 51.2869, Z -8.0000, A 0.000, B 0.000, C 0.000 }
gfCNCPoint6[403] = {X 32.5222, Y 52.1744, Z -8.0000, A 0.000, B 0.000, C 0.000 }
gfCNCPoint6[404] = {X 31.1566, Y 52.8874, Z -8.0000, A 0.000, B 0.000, C 0.000 }
gfCNCPoint6[405] = {X 29.7086, Y 53.4133, Z -8.0000, A 0.000, B 0.000, C 0.000 }
gfCNCPoint6[406] = {X 28.2038, Y 53.7429, Z -8.0000, A 0.000, B 0.000, C 0.000 }
gfCNCPoint6[407] = {X 26.6685, Y 53.8703, Z -8.0000, A 0.000, B 0.000, C 0.000 }
gfCNCPoint6[408] = {X 24.3197, Y 54.9131, Z -8.0000, A 0.000, B 0.000, C 0.000 }
gfCNCPoint6[409] = {X 21.9036, Y 55.7890, Z -8.0000, A 0.000, B 0.000, C 0.000 }
gfCNCPoint6[410] = {X 19.5299, Y 56.4649, Z -8.0000, A 0.000, B 0.000, C 0.000 }
gfCNCPoint6[411] = {X 17.1088, Y 56.9437, Z -8.0000, A 0.000, B 0.000, C 0.000 }
gfCNCPoint6[412] = {X 14.6565, Y 57.2220, Z -8.0000, A 0.000, B 0.000, C 0.000 }
gfCNCPoint6[413] = {X 12.1897, Y 57.2981, Z -8.0000, A 0.000, B 0.000, C 0.000 }
gfCNCPoint6[414] = {X 9.7249, Y 57.1713, Z -8.0000, A 0.000, B 0.000, C 0.000 }
gfCNCPoint6[415] = {X 8.4102, Y 57.0201, Z -8.0000, A 0.000, B 0.000, C 0.000 }
gfCNCPoint6[416] = {X 7.1033, Y 56.8111, Z -8.0000, A 0.000, B 0.000, C 0.000 }
gfCNCPoint6[417] = {X 7.1033, Y 92.8952, Z -8.0000, A 0.000, B 0.000, C 0.000 }
gfCNCPoint6[418] = {X 116.2646, Y 92.8952, Z -8.0000, A 0.000, B 0.000, C 0.000 }
gfCNCPoint6[419] = {X 116.9679, Y 91.6633, Z -8.0000, A 0.000, B 0.000, C 0.000 }
gfCNCPoint6[420] = {X 117.8438, Y 90.5475, Z -8.0000, A 0.000, B 0.000, C 0.000 }
gfCNCPoint6[421] = {X 118.8733, Y 89.5716, Z -8.0000, A 0.000, B 0.000, C 0.000 }
gfCNCPoint6[422] = {X 120.0343, Y 88.7566, Z -8.0000, A 0.000, B 0.000, C 0.000 }
gfCNCPoint6[423] = {X 121.3020, Y 88.1201, Z -8.0000, A 0.000, B 0.000, C 0.000 }
gfCNCPoint6[424] = {X 122.6491, Y 87.6757, Z -8.0000, A 0.000, B 0.000, C 0.000 }
gfCNCPoint6[425] = {X 124.0467, Y 87.4330, Z -8.0000, A 0.000, B 0.000, C 0.000 }
gfCNCPoint6[426] = {X 124.1412, Y 87.4182, Z -8.0000, A 0.000, B 0.000, C 0.000 }
gfCNCPoint6[427] = {X 124.5382, Y 87.3593, Z -8.0000, A 0.000, B 0.000, C 0.000 }
gfCNCPoint6[428] = {X 124.9951, Y 86.8918, Z -8.0000, A 0.000, B 0.000, C 0.000 }
gfCNCPoint6[429] = {X 125.4393, Y 86.4122, Z -8.0000, A 0.000, B 0.000, C 0.000 }
gfCNCPoint6[430] = {X 149.6584, Y 59.8181, Z -8.0000, A 0.000, B 0.000, C 0.000 }
gfCNCPoint6[431] = {X 149.6295, Y 59.4060, Z -8.0000, A 0.000, B 0.000, C 0.000 }
gfCNCPoint6[432] = {X 149.6181, Y 58.9930, Z -8.0000, A 0.000, B 0.000, C 0.000 }
gfCNCPoint6[433] = {X 149.6180, Y 58.0000, Z -8.0000, A 0.000, B 0.000, C 0.000 }
gfCNCPoint6[434] = {X 149.6915, Y 56.8093, Z -8.0000, A 0.000, B 0.000, C 0.000 }
gfCNCPoint6[435] = {X 149.9109, Y 55.6367, Z -8.0000, A 0.000, B 0.000, C 0.000 }
gfCNCPoint6[436] = {X 150.2729, Y 54.5000, Z -8.0000, A 0.000, B 0.000, C 0.000 }
gfCNCPoint6[437] = {X 150.7719, Y 53.4164, Z -8.0000, A 0.000, B 0.000, C 0.000 }
gfCNCPoint6[438] = {X 151.5117, Y 52.2488, Z -8.0000, A 0.000, B 0.000, C 0.000 }
gfCNCPoint6[439] = {X 152.4103, Y 51.1984, Z -8.0000, A 0.000, B 0.000, C 0.000 }
gfCNCPoint6[440] = {X 153.4493, Y 50.2867, Z -8.0000, A 0.000, B 0.000, C 0.000 }
gfCNCPoint6[441] = {X 154.6075, Y 49.5323, Z -8.0000, A 0.000, B 0.000, C 0.000 }
gfCNCPoint6[442] = {X 155.8614, Y 48.9505, Z -8.0000, A 0.000, B 0.000, C 0.000 }
gfCNCPoint6[443] = {X 157.1854, Y 48.5533, Z -8.0000, A 0.000, B 0.000, C 0.000 }
gfCNCPoint6[444] = {X 158.2353, Y 48.3785, Z -8.0000, A 0.000, B 0.000, C 0.000 }
gfCNCPoint6[445] = {X 159.2980, Y 48.3200, Z -8.0000, A 0.000, B 0.000, C 0.000 }
gfCNCPoint6[446] = {X 176.3030, Y 48.3200, Z -8.0000, A 0.000, B 0.000, C 0.000 }
gfCNCPoint6[447] = {X 174.9305, Y 47.4865, Z -8.0000, A 0.000, B 0.000, C 0.000 }
gfCNCPoint6[448] = {X 173.6417, Y 46.5286, Z -8.0000, A 0.000, B 0.000, C 0.000 }
gfCNCPoint6[449] = {X 172.5419, Y 45.5342, Z -8.0000, A 0.000, B 0.000, C 0.000 }
gfCNCPoint6[450] = {X 171.5570, Y 44.4260, Z -8.0000, A 0.000, B 0.000, C 0.000 }
gfCNCPoint6[451] = {X 170.5955, Y 43.0508, Z -8.0000, A 0.000, B 0.000, C 0.000 }
gfCNCPoint6[452] = {X 169.8108, Y 41.5676, Z -8.0000, A 0.000, B 0.000, C 0.000 }
gfCNCPoint6[453] = {X 169.2149, Y 39.9990, Z -8.0000, A 0.000, B 0.000, C 0.000 }
gfCNCPoint6[454] = {X 168.8169, Y 38.3690, Z -8.0000, A 0.000, B 0.000, C 0.000 }
gfCNCPoint6[455] = {X 168.7067, Y 37.6766, Z -8.0000, A 0.000, B 0.000, C 0.000 }
gfCNCPoint6[456] = {X 168.5417, Y 36.0106, Z -8.0000, A 0.000, B 0.000, C 0.000 }
gfCNCPoint6[457] = {X 168.5589, Y 34.3364, Z -8.0000, A 0.000, B 0.000, C 0.000 }
gfCNCPoint6[458] = {X 168.7583, Y 32.6741, Z -8.0000, A 0.000, B 0.000, C 0.000 }
gfCNCPoint6[459] = {X 169.1373, Y 31.0433, Z -8.0000, A 0.000, B 0.000, C 0.000 }
gfCNCPoint6[460] = {X 169.6915, Y 29.4635, Z -8.0000, A 0.000, B 0.000, C 0.000 }
gfCNCPoint6[461] = {X 170.2632, Y 28.2667, Z -8.0000, A 0.000, B 0.000, C 0.000 }
gfCNCPoint6[462] = {X 170.9699, Y 27.1444, Z -8.0000, A 0.000, B 0.000, C 0.000 }
gfCNCPoint6[463] = {X 171.8021, Y 26.1117, Z -8.0000, A 0.000, B 0.000, C 0.000 }
gfCNCPoint6[464] = {X 172.7485, Y 25.1825, Z -8.0000, A 0.000, B 0.000, C 0.000 }
gfCNCPoint6[465] = {X 173.7963, Y 24.3693, Z -8.0000, A 0.000, B 0.000, C 0.000 }
gfCNCPoint6[466] = {X 173.0265, Y 23.7512, Z -8.0000, A 0.000, B 0.000, C 0.000 }
gfCNCPoint6[467] = {X 172.3969, Y 22.9908, Z -8.0000, A 0.000, B 0.000, C 0.000 }
gfCNCPoint6[468] = {X 171.9332, Y 22.1193, Z -8.0000, A 0.000, B 0.000, C 0.000 }
gfCNCPoint6[469] = {X 169.3220, Y 15.7237, Z -8.0000, A 0.000, B 0.000, C 0.000 }
gfCNCPoint6[470] = {X 169.1088, Y 15.0753, Z -8.0000, A 0.000, B 0.000, C 0.000 }
gfCNCPoint6[471] = {X 168.9882, Y 14.4035, Z -8.0000, A 0.000, B 0.000, C 0.000 }
gfCNCPoint6[472] = {X 168.9599, Y 13.8791, Z -8.0000, A 0.000, B 0.000, C 0.000 }
gfCNCPoint6[473] = {X 168.9882, Y 13.3548, Z -8.0000, A 0.000, B 0.000, C 0.000 }
gfCNCPoint6[474] = {X 169.1590, Y 12.4994, Z -8.0000, A 0.000, B 0.000, C 0.000 }
gfCNCPoint6[475] = {X 169.4794, Y 11.6882, Z -8.0000, A 0.000, B 0.000, C 0.000 }
gfCNCPoint6[476] = {X 169.9391, Y 10.9469, Z -8.0000, A 0.000, B 0.000, C 0.000 }
gfCNCPoint6[477] = {X 170.6136, Y 10.2178, Z -8.0000, A 0.000, B 0.000, C 0.000 }
gfCNCPoint6[478] = {X 171.4217, Y 9.6404, Z -8.0000, A 0.000, B 0.000, C 0.000 }
gfCNCPoint6[479] = {X 172.0576, Y 9.2779, Z -8.0000, A 0.000, B 0.000, C 0.000 }
gfCNCPoint6[480] = {X 172.9923, Y 8.8772, Z -8.0000, A 0.000, B 0.000, C 0.000 }
gfCNCPoint6[481] = {X 173.9898, Y 8.6790, Z -8.0000, A 0.000, B 0.000, C 0.000 }
gfCNCPoint6[482] = {X 175.0067, Y 8.6918, Z -8.0000, A 0.000, B 0.000, C 0.000 }
gfCNCPoint6[483] = {X 175.9989, Y 8.9151, Z -8.0000, A 0.000, B 0.000, C 0.000 }
gfCNCPoint6[484] = {X 176.9082, Y 8.5286, Z -8.0000, A 0.000, B 0.000, C 0.000 }
gfCNCPoint6[485] = {X 179.1577, Y 7.7024, Z -8.0000, A 0.000, B 0.000, C 0.000 }
gfCNCPoint6[486] = {X 181.4784, Y 7.1048, Z -8.0000, A 0.000, B 0.000, C 0.000 }
gfCNCPoint6[487] = {X 168.0207, Y 7.1048, Z -8.0000, A 0.000, B 0.000, C 0.000 }
gfCNCPoint6[488] = {X 168.0207, Y 4.7048, Z -8.0000, A 0.000, B 0.000, C 0.000 }
gfCNCPoint6[489] = {X 155.1592, Y 4.7048, Z -8.0000, A 0.000, B 0.000, C 0.000 }
gfCNCPoint6[490] = {X 155.1592, Y 7.1048, Z -8.0000, A 0.000, B 0.000, C 0.000 }
gfCNCPoint6[491] = {X 137.3635, Y 7.1048, Z -8.0000, A 0.000, B 0.000, C 0.000 }
gfCNCPoint6[492] = {X 137.5329, Y 7.2907, Z -8.0000, A 0.000, B 0.000, C 0.000 }
gfCNCPoint6[493] = {X 137.6924, Y 7.4850, Z -8.0000, A 0.000, B 0.000, C 0.000 }
gfCNCPoint6[494] = {X 154.8303, Y 7.4850, Z -8.0000, A 0.000, B 0.000, C 0.000 }
gfCNCPoint6[495] = {X 154.9899, Y 7.2907, Z -8.0000, A 0.000, B 0.000, C 0.000 }
gfCNCPoint6[496] = {X 155.1592, Y 7.1048, Z -8.0000, A 0.000, B 0.000, C 0.000 }
gfCNCPoint6[497] = {X 155.1592, Y 4.7048, Z -8.0000, A 0.000, B 0.000, C 0.000 }
gfCNCPoint6[498] = {X 23.8402, Y 4.7048, Z -8.0000, A 0.000, B 0.000, C 0.000 }
gfCNCPoint6[499] = {X 25.7675, Y 5.7852, Z -8.0000, A 0.000, B 0.000, C 0.000 }
gfCNCPoint6[500] = {X 27.5783, Y 7.0510, Z -8.0000, A 0.000, B 0.000, C 0.000 }
gfCNCPoint6[501] = {X 28.5607, Y 7.8751, Z -8.0000, A 0.000, B 0.000, C 0.000 }
gfCNCPoint6[502] = {X 29.4815, Y 8.7674, Z -8.0000, A 0.000, B 0.000, C 0.000 }
gfCNCPoint6[503] = {X 30.6897, Y 10.1627, Z -8.0000, A 0.000, B 0.000, C 0.000 }
gfCNCPoint6[504] = {X 31.7477, Y 11.6752, Z -8.0000, A 0.000, B 0.000, C 0.000 }
gfCNCPoint6[505] = {X 32.6442, Y 13.2886, Z -8.0000, A 0.000, B 0.000, C 0.000 }
gfCNCPoint6[506] = {X 33.3696, Y 14.9859, Z -8.0000, A 0.000, B 0.000, C 0.000 }
gfCNCPoint6[507] = {X 33.9196, Y 16.8169, Z -8.0000, A 0.000, B 0.000, C 0.000 }
gfCNCPoint6[508] = {X 34.2912, Y 18.6923, Z -8.0000, A 0.000, B 0.000, C 0.000 }
gfCNCPoint6[509] = {X 34.4810, Y 20.5947, Z -8.0000, A 0.000, B 0.000, C 0.000 }
gfCNCPoint6[510] = {X 34.4873, Y 22.5065, Z -8.0000, A 0.000, B 0.000, C 0.000 }
gfCNCPoint6[511] = {X 34.3100, Y 24.4102, Z -8.0000, A 0.000, B 0.000, C 0.000 }
gfCNCPoint6[512] = {X 33.9507, Y 26.2879, Z -8.0000, A 0.000, B 0.000, C 0.000 }
gfCNCPoint6[513] = {X 33.4666, Y 27.9397, Z -8.0000, A 0.000, B 0.000, C 0.000 }
gfCNCPoint6[514] = {X 32.8139, Y 29.5324, Z -8.0000, A 0.000, B 0.000, C 0.000 }
gfCNCPoint6[515] = {X 31.9995, Y 31.0488, Z -8.0000, A 0.000, B 0.000, C 0.000 }
gfCNCPoint6[516] = {X 32.1288, Y 31.2843, Z -8.0000, A 0.000, B 0.000, C 0.000 }
gfCNCPoint6[517] = {X 32.2511, Y 31.5234, Z -8.0000, A 0.000, B 0.000, C 0.000 }
gfCNCPoint6[518] = {X 35.3025, Y 37.8269, Z -8.0000, A 0.000, B 0.000, C 0.000 }
gfCNCPoint6[519] = {X 35.7263, Y 38.8573, Z -8.0000, A 0.000, B 0.000, C 0.000 }
gfCNCPoint6[520] = {X 36.0224, Y 39.9313, Z -8.0000, A 0.000, B 0.000, C 0.000 }
gfCNCPoint6[521] = {X 36.1865, Y 41.0332, Z -8.0000, A 0.000, B 0.000, C 0.000 }
gfCNCPoint6[522] = {X 36.2163, Y 42.1469, Z -8.0000, A 0.000, B 0.000, C 0.000 }
gfCNCPoint6[523] = {X 36.6301, Y 41.4266, Z -8.0000, A 0.000, B 0.000, C 0.000 }
gfCNCPoint6[524] = {X 37.1601, Y 40.7868, Z -8.0000, A 0.000, B 0.000, C 0.000 }
gfCNCPoint6[525] = {X 37.7910, Y 40.2463, Z -8.0000, A 0.000, B 0.000, C 0.000 }
gfCNCPoint6[526] = {X 38.5044, Y 39.8205, Z -8.0000, A 0.000, B 0.000, C 0.000 }
gfCNCPoint6[527] = {X 39.0433, Y 38.5344, Z -8.0000, A 0.000, B 0.000, C 0.000 }
gfCNCPoint6[528] = {X 39.5393, Y 37.2311, Z -8.0000, A 0.000, B 0.000, C 0.000 }
gfCNCPoint6[529] = {X 47.6702, Y 15.4045, Z -8.0000, A 0.000, B 0.000, C 0.000 }
gfCNCPoint6[530] = {X 47.3200, Y 14.6512, Z -8.0000, A 0.000, B 0.000, C 0.000 }
gfCNCPoint6[531] = {X 47.1026, Y 13.8493, Z -8.0000, A 0.000, B 0.000, C 0.000 }
gfCNCPoint6[532] = {X 47.0244, Y 13.0222, Z -8.0000, A 0.000, B 0.000, C 0.000 }
gfCNCPoint6[533] = {X 47.0242, Y 12.1868, Z -8.0000, A 0.000, B 0.000, C 0.000 }
gfCNCPoint6[534] = {X 47.0722, Y 11.5041, Z -8.0000, A 0.000, B 0.000, C 0.000 }
gfCNCPoint6[535] = {X 47.2153, Y 10.8347, Z -8.0000, A 0.000, B 0.000, C 0.000 }
gfCNCPoint6[536] = {X 42.6032, Y 9.5048, Z -8.0000, A 0.000, B 0.000, C 0.000 }
gfCNCPoint6[537] = {X 36.0467, Y 9.5048, Z -8.0000, A 0.000, B 0.000, C 0.000 }
gfCNCPoint6[538] = {X 37.0568, Y 11.3879, Z -8.0000, A 0.000, B 0.000, C 0.000 }
gfCNCPoint6[539] = {X 37.8852, Y 13.3577, Z -8.0000, A 0.000, B 0.000, C 0.000 }
gfCNCPoint6[540] = {X 38.5474, Y 15.5379, Z -8.0000, A 0.000, B 0.000, C 0.000 }
gfCNCPoint6[541] = {X 39.0058, Y 17.7698, Z -8.0000, A 0.000, B 0.000, C 0.000 }
gfCNCPoint6[542] = {X 39.2566, Y 20.0345, Z -8.0000, A 0.000, B 0.000, C 0.000 }
gfCNCPoint6[543] = {X 39.2974, Y 22.3126, Z -8.0000, A 0.000, B 0.000, C 0.000 }
gfCNCPoint6[544] = {X 39.1281, Y 24.5848, Z -8.0000, A 0.000, B 0.000, C 0.000 }
gfCNCPoint6[545] = {X 42.5393, Y 15.4278, Z -8.0000, A 0.000, B 0.000, C 0.000 }
gfCNCPoint6[546] = {X 42.3075, Y 14.2451, Z -8.0000, A 0.000, B 0.000, C 0.000 }
gfCNCPoint6[547] = {X 42.2244, Y 13.0428, Z -8.0000, A 0.000, B 0.000, C 0.000 }
gfCNCPoint6[548] = {X 42.2242, Y 12.1868, Z -8.0000, A 0.000, B 0.000, C 0.000 }
gfCNCPoint6[549] = {X 42.3194, Y 10.8325, Z -8.0000, A 0.000, B 0.000, C 0.000 }
gfCNCPoint6[550] = {X 42.6032, Y 9.5048, Z -8.0000, A 0.000, B 0.000, C 0.000 }
gfCNCPoint6[551] = {X 44.9092, Y 10.1698, Z -8.0000, A 0.000, B 0.000, C 0.000 }
gfCNCPoint6[552] = {X 45.3324, Y 9.0549, Z -8.0000, A 0.000, B 0.000, C 0.000 }
gfCNCPoint6[553] = {X 45.9318, Y 8.0240, Z -8.0000, A 0.000, B 0.000, C 0.000 }
gfCNCPoint6[554] = {X 46.6916, Y 7.1048, Z -8.0000, A 0.000, B 0.000, C 0.000 }
gfCNCPoint6[555] = {X 31.2124, Y 7.1048, Z -8.0000, A 0.000, B 0.000, C 0.000 }
gfCNCPoint6[556] = {X 32.2278, Y 8.2449, Z -8.0000, A 0.000, B 0.000, C 0.000 }
gfCNCPoint6[557] = {X 33.1546, Y 9.4581, Z -8.0000, A 0.000, B 0.000, C 0.000 }
gfCNCPoint6[558] = {X 33.9875, Y 10.7376, Z -8.0000, A 0.000, B 0.000, C 0.000 }
gfCNCPoint6[559] = {X 34.8882, Y 12.4161, Z -8.0000, A 0.000, B 0.000, C 0.000 }
gfCNCPoint6[560] = {X 35.6274, Y 14.1718, Z -8.0000, A 0.000, B 0.000, C 0.000 }
gfCNCPoint6[561] = {X 36.2236, Y 16.1380, Z -8.0000, A 0.000, B 0.000, C 0.000 }
gfCNCPoint6[562] = {X 36.6362, Y 18.1507, Z -8.0000, A 0.000, B 0.000, C 0.000 }
gfCNCPoint6[563] = {X 36.8618, Y 20.1930, Z -8.0000, A 0.000, B 0.000, C 0.000 }
gfCNCPoint6[564] = {X 36.8983, Y 22.2473, Z -8.0000, A 0.000, B 0.000, C 0.000 }
gfCNCPoint6[565] = {X 36.7455, Y 24.2962, Z -8.0000, A 0.000, B 0.000, C 0.000 }
gfCNCPoint6[566] = {X 36.5522, Y 25.5784, Z -8.0000, A 0.000, B 0.000, C 0.000 }
gfCNCPoint6[567] = {X 36.2847, Y 26.8471, Z -8.0000, A 0.000, B 0.000, C 0.000 }
gfCNCPoint6[568] = {X 35.8755, Y 28.3066, Z -8.0000, A 0.000, B 0.000, C 0.000 }
gfCNCPoint6[569] = {X 35.3511, Y 29.7289, Z -8.0000, A 0.000, B 0.000, C 0.000 }
gfCNCPoint6[570] = {X 34.7149, Y 31.1047, Z -8.0000, A 0.000, B 0.000, C 0.000 }
gfCNCPoint6[571] = {X 37.2836, Y 36.4113, Z -8.0000, A 0.000, B 0.000, C 0.000 }
gfCNCPoint6[572] = {X 41.3771, Y 25.4226, Z -8.0000, A 0.000, B 0.000, C 0.000 }
gfCNCPoint6[573] = {X 45.0743, Y 15.4980, Z -8.0000, A 0.000, B 0.000, C 0.000 }
gfCNCPoint6[574] = {X 44.7425, Y 14.2852, Z -8.0000, A 0.000, B 0.000, C 0.000 }
gfCNCPoint6[575] = {X 44.6244, Y 13.0334, Z -8.0000, A 0.000, B 0.000, C 0.000 }
gfCNCPoint6[576] = {X 44.6242, Y 12.1868, Z -8.0000, A 0.000, B 0.000, C 0.000 }
gfCNCPoint6[577] = {X 44.6958, Y 11.1683, Z -8.0000, A 0.000, B 0.000, C 0.000 }
gfCNCPoint6[578] = {X 44.9092, Y 10.1698, Z -8.0000, A 0.000, B 0.000, C 0.000 }
gfCNCPoint6[579] = {X 47.2153, Y 10.8347, Z -8.0000, A 0.000, B 0.000, C 0.000 }
gfCNCPoint6[580] = {X 47.4989, Y 10.0874, Z -8.0000, A 0.000, B 0.000, C 0.000 }
gfCNCPoint6[581] = {X 47.9008, Y 9.3964, Z -8.0000, A 0.000, B 0.000, C 0.000 }
gfCNCPoint6[582] = {X 48.4100, Y 8.7802, Z -8.0000, A 0.000, B 0.000, C 0.000 }
gfCNCPoint6[583] = {X 49.1545, Y 8.1552, Z -8.0000, A 0.000, B 0.000, C 0.000 }
gfCNCPoint6[584] = {X 50.0082, Y 7.6902, Z -8.0000, A 0.000, B 0.000, C 0.000 }
gfCNCPoint6[585] = {X 50.9370, Y 7.4036, Z -8.0000, A 0.000, B 0.000, C 0.000 }
gfCNCPoint6[586] = {X 51.9042, Y 7.3068, Z -8.0000, A 0.000, B 0.000, C 0.000 }
gfCNCPoint6[587] = {X 59.6221, Y 7.3068, Z -8.0000, A 0.000, B 0.000, C 0.000 }
gfCNCPoint6[588] = {X 60.5893, Y 7.4036, Z -8.0000, A 0.000, B 0.000, C 0.000 }
gfCNCPoint6[589] = {X 61.5182, Y 7.6902, Z -8.0000, A 0.000, B 0.000, C 0.000 }
gfCNCPoint6[590] = {X 62.3718, Y 8.1552, Z -8.0000, A 0.000, B 0.000, C 0.000 }
gfCNCPoint6[591] = {X 63.1163, Y 8.7802, Z -8.0000, A 0.000, B 0.000, C 0.000 }
gfCNCPoint6[592] = {X 63.7053, Y 9.5144, Z -8.0000, A 0.000, B 0.000, C 0.000 }
gfCNCPoint6[593] = {X 64.1424, Y 10.3480, Z -8.0000, A 0.000, B 0.000, C 0.000 }
gfCNCPoint6[594] = {X 64.4114, Y 11.2500, Z -8.0000, A 0.000, B 0.000, C 0.000 }
gfCNCPoint6[595] = {X 64.5021, Y 12.1868, Z -8.0000, A 0.000, B 0.000, C 0.000 }
gfCNCPoint6[596] = {X 64.5019, Y 13.0237, Z -8.0000, A 0.000, B 0.000, C 0.000 }
gfCNCPoint6[597] = {X 64.4205, Y 13.8669, Z -8.0000, A 0.000, B 0.000, C 0.000 }
gfCNCPoint6[598] = {X 64.1944, Y 14.6834, Z -8.0000, A 0.000, B 0.000, C 0.000 }
gfCNCPoint6[599] = {X 63.8306, Y 15.4484, Z -8.0000, A 0.000, B 0.000, C 0.000 }
gfCNCPoint6[600] = {X 72.9561, Y 39.8587, Z -8.0000, A 0.000, B 0.000, C 0.000 }
gfCNCPoint6[601] = {X 73.8455, Y 40.4408, Z -8.0000, A 0.000, B 0.000, C 0.000 }
gfCNCPoint6[602] = {X 74.5878, Y 41.2017, Z -8.0000, A 0.000, B 0.000, C 0.000 }
gfCNCPoint6[603] = {X 75.1478, Y 42.1052, Z -8.0000, A 0.000, B 0.000, C 0.000 }
gfCNCPoint6[604] = {X 75.4988, Y 43.1085, Z -8.0000, A 0.000, B 0.000, C 0.000 }
gfCNCPoint6[605] = {X 75.6243, Y 44.1640, Z -8.0000, A 0.000, B 0.000, C 0.000 }
gfCNCPoint6[606] = {X 75.6245, Y 45.0000, Z -8.0000, A 0.000, B 0.000, C 0.000 }
gfCNCPoint6[607] = {X 75.5307, Y 45.9520, Z -8.0000, A 0.000, B 0.000, C 0.000 }
gfCNCPoint6[608] = {X 75.2530, Y 46.8675, Z -8.0000, A 0.000, B 0.000, C 0.000 }
gfCNCPoint6[609] = {X 74.8020, Y 47.7112, Z -8.0000, A 0.000, B 0.000, C 0.000 }
gfCNCPoint6[610] = {X 74.1951, Y 48.4507, Z -8.0000, A 0.000, B 0.000, C 0.000 }
gfCNCPoint6[611] = {X 73.4556, Y 49.0576, Z -8.0000, A 0.000, B 0.000, C 0.000 }
gfCNCPoint6[612] = {X 72.6120, Y 49.5085, Z -8.0000, A 0.000, B 0.000, C 0.000 }
gfCNCPoint6[613] = {X 71.6965, Y 49.7862, Z -8.0000, A 0.000, B 0.000, C 0.000 }
gfCNCPoint6[614] = {X 70.7445, Y 49.8800, Z -8.0000, A 0.000, B 0.000, C 0.000 }
gfCNCPoint6[615] = {X 64.1851, Y 49.8800, Z -8.0000, A 0.000, B 0.000, C 0.000 }
gfCNCPoint6[616] = {X 63.2331, Y 49.7862, Z -8.0000, A 0.000, B 0.000, C 0.000 }
gfCNCPoint6[617] = {X 62.3176, Y 49.5085, Z -8.0000, A 0.000, B 0.000, C 0.000 }
gfCNCPoint6[618] = {X 61.4740, Y 49.0576, Z -8.0000, A 0.000, B 0.000, C 0.000 }
gfCNCPoint6[619] = {X 60.7345, Y 48.4507, Z -8.0000, A 0.000, B 0.000, C 0.000 }
gfCNCPoint6[620] = {X 60.1276, Y 47.7112, Z -8.0000, A 0.000, B 0.000, C 0.000 }
gfCNCPoint6[621] = {X 59.6766, Y 46.8675, Z -8.0000, A 0.000, B 0.000, C 0.000 }
gfCNCPoint6[622] = {X 59.3989, Y 45.9520, Z -8.0000, A 0.000, B 0.000, C 0.000 }
gfCNCPoint6[623] = {X 59.3051, Y 45.0000, Z -8.0000, A 0.000, B 0.000, C 0.000 }
gfCNCPoint6[624] = {X 59.3052, Y 44.2028, Z -8.0000, A 0.000, B 0.000, C 0.000 }
gfCNCPoint6[625] = {X 59.3846, Y 43.3315, Z -8.0000, A 0.000, B 0.000, C 0.000 }
gfCNCPoint6[626] = {X 59.6184, Y 42.4884, Z -8.0000, A 0.000, B 0.000, C 0.000 }
gfCNCPoint6[627] = {X 59.9990, Y 41.7006, Z -8.0000, A 0.000, B 0.000, C 0.000 }
gfCNCPoint6[628] = {X 59.6148, Y 40.6492, Z -8.0000, A 0.000, B 0.000, C 0.000 }
gfCNCPoint6[629] = {X 52.4676, Y 40.6492, Z -8.0000, A 0.000, B 0.000, C 0.000 }
gfCNCPoint6[630] = {X 51.9477, Y 42.0463, Z -8.0000, A 0.000, B 0.000, C 0.000 }
gfCNCPoint6[631] = {X 52.2220, Y 42.7252, Z -8.0000, A 0.000, B 0.000, C 0.000 }
gfCNCPoint6[632] = {X 52.3916, Y 43.4375, Z -8.0000, A 0.000, B 0.000, C 0.000 }
gfCNCPoint6[633] = {X 52.4528, Y 44.1672, Z -8.0000, A 0.000, B 0.000, C 0.000 }
gfCNCPoint6[634] = {X 52.4529, Y 45.0000, Z -8.0000, A 0.000, B 0.000, C 0.000 }
gfCNCPoint6[635] = {X 52.3592, Y 45.9520, Z -8.0000, A 0.000, B 0.000, C 0.000 }
gfCNCPoint6[636] = {X 52.0815, Y 46.8675, Z -8.0000, A 0.000, B 0.000, C 0.000 }
gfCNCPoint6[637] = {X 51.6305, Y 47.7112, Z -8.0000, A 0.000, B 0.000, C 0.000 }
gfCNCPoint6[638] = {X 51.0236, Y 48.4507, Z -8.0000, A 0.000, B 0.000, C 0.000 }
gfCNCPoint6[639] = {X 50.2841, Y 49.0576, Z -8.0000, A 0.000, B 0.000, C 0.000 }
gfCNCPoint6[640] = {X 49.4404, Y 49.5085, Z -8.0000, A 0.000, B 0.000, C 0.000 }
gfCNCPoint6[641] = {X 48.5250, Y 49.7862, Z -8.0000, A 0.000, B 0.000, C 0.000 }
gfCNCPoint6[642] = {X 47.5729, Y 49.8800, Z -8.0000, A 0.000, B 0.000, C 0.000 }
gfCNCPoint6[643] = {X 40.6393, Y 49.8800, Z -8.0000, A 0.000, B 0.000, C 0.000 }
gfCNCPoint6[644] = {X 39.6433, Y 49.7773, Z -8.0000, A 0.000, B 0.000, C 0.000 }
gfCNCPoint6[645] = {X 38.6892, Y 49.4734, Z -8.0000, A 0.000, B 0.000, C 0.000 }
gfCNCPoint6[646] = {X 37.8173, Y 48.9813, Z -8.0000, A 0.000, B 0.000, C 0.000 }
gfCNCPoint6[647] = {X 37.0641, Y 48.3215, Z -8.0000, A 0.000, B 0.000, C 0.000 }
gfCNCPoint6[648] = {X 36.5085, Y 47.5983, Z -8.0000, A 0.000, B 0.000, C 0.000 }
gfCNCPoint6[649] = {X 36.0972, Y 46.7843, Z -8.0000, A 0.000, B 0.000, C 0.000 }
gfCNCPoint6[650] = {X 35.8445, Y 45.9080, Z -8.0000, A 0.000, B 0.000, C 0.000 }
gfCNCPoint6[651] = {X 35.7593, Y 45.0000, Z -8.0000, A 0.000, B 0.000, C 0.000 }
gfCNCPoint6[652] = {X 35.7593, Y 44.7148, Z -8.0000, A 0.000, B 0.000, C 0.000 }
gfCNCPoint6[653] = {X 36.2393, Y 44.7148, Z -8.0000, A 0.000, B 0.000, C 0.000 }
gfCNCPoint6[654] = {X 36.2397, Y 44.1483, Z -8.0000, A 0.000, B 0.000, C 0.000 }
gfCNCPoint6[655] = {X 36.3680, Y 43.1525, Z -8.0000, A 0.000, B 0.000, C 0.000 }
gfCNCPoint6[656] = {X 36.7186, Y 42.2118, Z -8.0000, A 0.000, B 0.000, C 0.000 }
gfCNCPoint6[657] = {X 37.2733, Y 41.3750, Z -8.0000, A 0.000, B 0.000, C 0.000 }
gfCNCPoint6[658] = {X 38.0033, Y 40.6858, Z -8.0000, A 0.000, B 0.000, C 0.000 }
gfCNCPoint6[659] = {X 38.8705, Y 40.1800, Z -8.0000, A 0.000, B 0.000, C 0.000 }
gfCNCPoint6[660] = {X 39.4543, Y 38.7992, Z -8.0000, A 0.000, B 0.000, C 0.000 }
gfCNCPoint6[661] = {X 39.9891, Y 37.3986, Z -8.0000, A 0.000, B 0.000, C 0.000 }
gfCNCPoint6[662] = {X 48.2011, Y 15.3544, Z -8.0000, A 0.000, B 0.000, C 0.000 }
gfCNCPoint6[663] = {X 47.8187, Y 14.6115, Z -8.0000, A 0.000, B 0.000, C 0.000 }
gfCNCPoint6[664] = {X 47.5835, Y 13.8097, Z -8.0000, A 0.000, B 0.000, C 0.000 }
gfCNCPoint6[665] = {X 47.5042, Y 12.9780, Z -8.0000, A 0.000, B 0.000, C 0.000 }
gfCNCPoint6[666] = {X 47.5042, Y 12.1868, Z -8.0000, A 0.000, B 0.000, C 0.000 }
gfCNCPoint6[667] = {X 47.6145, Y 11.2077, Z -8.0000, A 0.000, B 0.000, C 0.000 }
gfCNCPoint6[668] = {X 47.9400, Y 10.2777, Z -8.0000, A 0.000, B 0.000, C 0.000 }
gfCNCPoint6[669] = {X 48.4642, Y 9.4435, Z -8.0000, A 0.000, B 0.000, C 0.000 }
gfCNCPoint6[670] = {X 49.1609, Y 8.7468, Z -8.0000, A 0.000, B 0.000, C 0.000 }
gfCNCPoint6[671] = {X 49.9951, Y 8.2226, Z -8.0000, A 0.000, B 0.000, C 0.000 }
gfCNCPoint6[672] = {X 50.9251, Y 7.8971, Z -8.0000, A 0.000, B 0.000, C 0.000 }
gfCNCPoint6[673] = {X 51.9042, Y 7.7868, Z -8.0000, A 0.000, B 0.000, C 0.000 }
gfCNCPoint6[674] = {X 59.6221, Y 7.7868, Z -8.0000, A 0.000, B 0.000, C 0.000 }
gfCNCPoint6[675] = {X 60.6012, Y 7.8971, Z -8.0000, A 0.000, B 0.000, C 0.000 }
gfCNCPoint6[676] = {X 61.5312, Y 8.2226, Z -8.0000, A 0.000, B 0.000, C 0.000 }
gfCNCPoint6[677] = {X 62.3655, Y 8.7468, Z -8.0000, A 0.000, B 0.000, C 0.000 }
gfCNCPoint6[678] = {X 63.0622, Y 9.4435, Z -8.0000, A 0.000, B 0.000, C 0.000 }
gfCNCPoint6[679] = {X 63.5864, Y 10.2777, Z -8.0000, A 0.000, B 0.000, C 0.000 }
gfCNCPoint6[680] = {X 63.9118, Y 11.2077, Z -8.0000, A 0.000, B 0.000, C 0.000 }
gfCNCPoint6[681] = {X 64.0221, Y 12.1868, Z -8.0000, A 0.000, B 0.000, C 0.000 }
gfCNCPoint6[682] = {X 64.0219, Y 13.0233, Z -8.0000, A 0.000, B 0.000, C 0.000 }
gfCNCPoint6[683] = {X 63.9336, Y 13.8560, Z -8.0000, A 0.000, B 0.000, C 0.000 }
gfCNCPoint6[684] = {X 63.6893, Y 14.6568, Z -8.0000, A 0.000, B 0.000, C 0.000 }
gfCNCPoint6[685] = {X 63.2976, Y 15.3969, Z -8.0000, A 0.000, B 0.000, C 0.000 }
gfCNCPoint6[686] = {X 63.5021, Y 15.9354, Z -8.0000, A 0.000, B 0.000, C 0.000 }
gfCNCPoint6[687] = {X 66.3154, Y 23.4026, Z -8.0000, A 0.000, B 0.000, C 0.000 }
gfCNCPoint6[688] = {X 72.2857, Y 39.4717, Z -8.0000, A 0.000, B 0.000, C 0.000 }
gfCNCPoint6[689] = {X 72.5790, Y 40.2095, Z -8.0000, A 0.000, B 0.000, C 0.000 }
gfCNCPoint6[690] = {X 73.4360, Y 40.7281, Z -8.0000, A 0.000, B 0.000, C 0.000 }
gfCNCPoint6[691] = {X 74.1535, Y 41.4270, Z -8.0000, A 0.000, B 0.000, C 0.000 }
gfCNCPoint6[692] = {X 74.6943, Y 42.2701, Z -8.0000, A 0.000, B 0.000, C 0.000 }
gfCNCPoint6[693] = {X 75.0305, Y 43.2137, Z -8.0000, A 0.000, B 0.000, C 0.000 }
gfCNCPoint6[694] = {X 75.1445, Y 44.2089, Z -8.0000, A 0.000, B 0.000, C 0.000 }
gfCNCPoint6[695] = {X 75.1445, Y 45.0000, Z -8.0000, A 0.000, B 0.000, C 0.000 }
gfCNCPoint6[696] = {X 75.0341, Y 45.9791, Z -8.0000, A 0.000, B 0.000, C 0.000 }
gfCNCPoint6[697] = {X 74.7087, Y 46.9091, Z -8.0000, A 0.000, B 0.000, C 0.000 }
gfCNCPoint6[698] = {X 74.1845, Y 47.7434, Z -8.0000, A 0.000, B 0.000, C 0.000 }
gfCNCPoint6[699] = {X 73.4878, Y 48.4401, Z -8.0000, A 0.000, B 0.000, C 0.000 }
gfCNCPoint6[700] = {X 72.6535, Y 48.9643, Z -8.0000, A 0.000, B 0.000, C 0.000 }
gfCNCPoint6[701] = {X 71.7236, Y 49.2897, Z -8.0000, A 0.000, B 0.000, C 0.000 }
gfCNCPoint6[702] = {X 70.7445, Y 49.4000, Z -8.0000, A 0.000, B 0.000, C 0.000 }
gfCNCPoint6[703] = {X 64.1851, Y 49.4000, Z -8.0000, A 0.000, B 0.000, C 0.000 }
gfCNCPoint6[704] = {X 63.2060, Y 49.2897, Z -8.0000, A 0.000, B 0.000, C 0.000 }
gfCNCPoint6[705] = {X 62.2760, Y 48.9643, Z -8.0000, A 0.000, B 0.000, C 0.000 }
gfCNCPoint6[706] = {X 61.4418, Y 48.4401, Z -8.0000, A 0.000, B 0.000, C 0.000 }
gfCNCPoint6[707] = {X 60.7451, Y 47.7434, Z -8.0000, A 0.000, B 0.000, C 0.000 }
gfCNCPoint6[708] = {X 60.2209, Y 46.9091, Z -8.0000, A 0.000, B 0.000, C 0.000 }
gfCNCPoint6[709] = {X 59.8955, Y 45.9791, Z -8.0000, A 0.000, B 0.000, C 0.000 }
gfCNCPoint6[710] = {X 59.7851, Y 45.0000, Z -8.0000, A 0.000, B 0.000, C 0.000 }
gfCNCPoint6[711] = {X 59.7856, Y 44.1483, Z -8.0000, A 0.000, B 0.000, C 0.000 }
gfCNCPoint6[712] = {X 59.8783, Y 43.3083, Z -8.0000, A 0.000, B 0.000, C 0.000 }
gfCNCPoint6[713] = {X 60.1298, Y 42.5016, Z -8.0000, A 0.000, B 0.000, C 0.000 }
gfCNCPoint6[714] = {X 60.5310, Y 41.7578, Z -8.0000, A 0.000, B 0.000, C 0.000 }
gfCNCPoint6[715] = {X 59.9504, Y 40.1692, Z -8.0000, A 0.000, B 0.000, C 0.000 }
gfCNCPoint6[716] = {X 52.1341, Y 40.1692, Z -8.0000, A 0.000, B 0.000, C 0.000 }
gfCNCPoint6[717] = {X 51.4233, Y 42.0792, Z -8.0000, A 0.000, B 0.000, C 0.000 }
gfCNCPoint6[718] = {X 51.7257, Y 42.7547, Z -8.0000, A 0.000, B 0.000, C 0.000 }
gfCNCPoint6[719] = {X 51.9107, Y 43.4714, Z -8.0000, A 0.000, B 0.000, C 0.000 }
gfCNCPoint6[720] = {X 51.9729, Y 44.2089, Z -8.0000, A 0.000, B 0.000, C 0.000 }
gfCNCPoint6[721] = {X 51.9729, Y 45.0000, Z -8.0000, A 0.000, B 0.000, C 0.000 }
gfCNCPoint6[722] = {X 51.8626, Y 45.9791, Z -8.0000, A 0.000, B 0.000, C 0.000 }
gfCNCPoint6[723] = {X 51.5372, Y 46.9091, Z -8.0000, A 0.000, B 0.000, C 0.000 }
gfCNCPoint6[724] = {X 51.0130, Y 47.7434, Z -8.0000, A 0.000, B 0.000, C 0.000 }
gfCNCPoint6[725] = {X 50.3163, Y 48.4401, Z -8.0000, A 0.000, B 0.000, C 0.000 }
gfCNCPoint6[726] = {X 49.4820, Y 48.9643, Z -8.0000, A 0.000, B 0.000, C 0.000 }
gfCNCPoint6[727] = {X 48.5520, Y 49.2897, Z -8.0000, A 0.000, B 0.000, C 0.000 }
gfCNCPoint6[728] = {X 47.5729, Y 49.4000, Z -8.0000, A 0.000, B 0.000, C 0.000 }
gfCNCPoint6[729] = {X 40.6393, Y 49.4000, Z -8.0000, A 0.000, B 0.000, C 0.000 }
gfCNCPoint6[730] = {X 39.6602, Y 49.2897, Z -8.0000, A 0.000, B 0.000, C 0.000 }
gfCNCPoint6[731] = {X 38.7302, Y 48.9643, Z -8.0000, A 0.000, B 0.000, C 0.000 }
gfCNCPoint6[732] = {X 37.8959, Y 48.4401, Z -8.0000, A 0.000, B 0.000, C 0.000 }
gfCNCPoint6[733] = {X 37.1992, Y 47.7434, Z -8.0000, A 0.000, B 0.000, C 0.000 }
gfCNCPoint6[734] = {X 36.6750, Y 46.9091, Z -8.0000, A 0.000, B 0.000, C 0.000 }
gfCNCPoint6[735] = {X 36.3496, Y 45.9791, Z -8.0000, A 0.000, B 0.000, C 0.000 }
gfCNCPoint6[736] = {X 36.2393, Y 45.0000, Z -8.0000, A 0.000, B 0.000, C 0.000 }
gfCNCPoint6[737] = {X 36.2393, Y 44.7148, Z -8.0000, A 0.000, B 0.000, C 0.000 }
gfCNCPoint6[738] = {X 35.7593, Y 44.7148, Z -8.0000, A 0.000, B 0.000, C 0.000 }
gfCNCPoint6[739] = {X 35.2211, Y 46.0074, Z -8.0000, A 0.000, B 0.000, C 0.000 }
gfCNCPoint6[740] = {X 34.4930, Y 47.2034, Z -8.0000, A 0.000, B 0.000, C 0.000 }
gfCNCPoint6[741] = {X 33.5918, Y 48.2750, Z -8.0000, A 0.000, B 0.000, C 0.000 }
gfCNCPoint6[742] = {X 33.2092, Y 48.6435, Z -8.0000, A 0.000, B 0.000, C 0.000 }
gfCNCPoint6[743] = {X 32.8060, Y 48.9892, Z -8.0000, A 0.000, B 0.000, C 0.000 }
gfCNCPoint6[744] = {X 32.2716, Y 49.4213, Z -8.0000, A 0.000, B 0.000, C 0.000 }
gfCNCPoint6[745] = {X 31.1849, Y 50.1782, Z -8.0000, A 0.000, B 0.000, C 0.000 }
gfCNCPoint6[746] = {X 30.0009, Y 50.7715, Z -8.0000, A 0.000, B 0.000, C 0.000 }
gfCNCPoint6[747] = {X 28.7440, Y 51.1887, Z -8.0000, A 0.000, B 0.000, C 0.000 }
gfCNCPoint6[748] = {X 27.4403, Y 51.4214, Z -8.0000, A 0.000, B 0.000, C 0.000 }
gfCNCPoint6[749] = {X 26.1167, Y 51.4647, Z -8.0000, A 0.000, B 0.000, C 0.000 }
gfCNCPoint6[750] = {X 23.6776, Y 52.5832, Z -8.0000, A 0.000, B 0.000, C 0.000 }
gfCNCPoint6[751] = {X 21.1585, Y 53.5075, Z -8.0000, A 0.000, B 0.000, C 0.000 }
gfCNCPoint6[752] = {X 18.9470, Y 54.1367, Z -8.0000, A 0.000, B 0.000, C 0.000 }
gfCNCPoint6[753] = {X 16.6908, Y 54.5798, Z -8.0000, A 0.000, B 0.000, C 0.000 }
gfCNCPoint6[754] = {X 14.4056, Y 54.8337, Z -8.0000, A 0.000, B 0.000, C 0.000 }
gfCNCPoint6[755] = {X 12.1072, Y 54.8969, Z -8.0000, A 0.000, B 0.000, C 0.000 }
gfCNCPoint6[756] = {X 9.8115, Y 54.7687, Z -8.0000, A 0.000, B 0.000, C 0.000 }
gfCNCPoint6[757] = {X 7.5344, Y 54.4501, Z -8.0000, A 0.000, B 0.000, C 0.000 }
gfCNCPoint6[758] = {X 7.1095, Y 54.3691, Z -8.0000, A 0.000, B 0.000, C 0.000 }
gfCNCPoint6[759] = {X 6.6859, Y 54.2814, Z -8.0000, A 0.000, B 0.000, C 0.000 }
gfCNCPoint6[760] = {X 5.6884, Y 54.0452, Z -8.0000, A 0.000, B 0.000, C 0.000 }
gfCNCPoint6[761] = {X 4.7033, Y 53.7619, Z -8.0000, A 0.000, B 0.000, C 0.000 }
gfCNCPoint6[762] = {X 4.7033, Y 95.2952, Z -8.0000, A 0.000, B 0.000, C 0.000 }
gfCNCPoint6[763] = {X 117.9386, Y 95.2952, Z -8.0000, A 0.000, B 0.000, C 0.000 }
gfCNCPoint6[764] = {X 118.3603, Y 94.0805, Z -8.0000, A 0.000, B 0.000, C 0.000 }
gfCNCPoint6[765] = {X 118.9891, Y 92.9589, Z -8.0000, A 0.000, B 0.000, C 0.000 }
gfCNCPoint6[766] = {X 119.8054, Y 91.9655, Z -8.0000, A 0.000, B 0.000, C 0.000 }
gfCNCPoint6[767] = {X 120.7838, Y 91.1311, Z -8.0000, A 0.000, B 0.000, C 0.000 }
gfCNCPoint6[768] = {X 121.8937, Y 90.4819, Z -8.0000, A 0.000, B 0.000, C 0.000 }
gfCNCPoint6[769] = {X 123.1004, Y 90.0381, Z -8.0000, A 0.000, B 0.000, C 0.000 }
gfCNCPoint6[770] = {X 124.3665, Y 89.8136, Z -8.0000, A 0.000, B 0.000, C 0.000 }
gfCNCPoint6[771] = {X 124.4298, Y 89.8022, Z -8.0000, A 0.000, B 0.000, C 0.000 }
gfCNCPoint6[772] = {X 124.4934, Y 89.7922, Z -8.0000, A 0.000, B 0.000, C 0.000 }
gfCNCPoint6[773] = {X 125.0303, Y 89.7125, Z -8.0000, A 0.000, B 0.000, C 0.000 }
gfCNCPoint6[774] = {X 125.3492, Y 89.6651, Z -8.0000, A 0.000, B 0.000, C 0.000 }
gfCNCPoint6[775] = {X 125.6663, Y 89.6069, Z -8.0000, A 0.000, B 0.000, C 0.000 }
gfCNCPoint6[776] = {X 126.4583, Y 88.8315, Z -8.0000, A 0.000, B 0.000, C 0.000 }
gfCNCPoint6[777] = {X 127.2176, Y 88.0240, Z -8.0000, A 0.000, B 0.000, C 0.000 }
gfCNCPoint6[778] = {X 152.2073, Y 60.5836, Z -8.0000, A 0.000, B 0.000, C 0.000 }
gfCNCPoint6[779] = {X 152.0684, Y 59.7893, Z -8.0000, A 0.000, B 0.000, C 0.000 }
gfCNCPoint6[780] = {X 152.0181, Y 58.9845, Z -8.0000, A 0.000, B 0.000, C 0.000 }
gfCNCPoint6[781] = {X 152.0180, Y 58.0000, Z -8.0000, A 0.000, B 0.000, C 0.000 }
gfCNCPoint6[782] = {X 152.1286, Y 56.7358, Z -8.0000, A 0.000, B 0.000, C 0.000 }
gfCNCPoint6[783] = {X 152.4570, Y 55.5101, Z -8.0000, A 0.000, B 0.000, C 0.000 }
gfCNCPoint6[784] = {X 152.9933, Y 54.3600, Z -8.0000, A 0.000, B 0.000, C 0.000 }
gfCNCPoint6[785] = {X 153.7212, Y 53.3205, Z -8.0000, A 0.000, B 0.000, C 0.000 }
gfCNCPoint6[786] = {X 154.6185, Y 52.4232, Z -8.0000, A 0.000, B 0.000, C 0.000 }
gfCNCPoint6[787] = {X 155.6580, Y 51.6953, Z -8.0000, A 0.000, B 0.000, C 0.000 }
gfCNCPoint6[788] = {X 156.8081, Y 51.1590, Z -8.0000, A 0.000, B 0.000, C 0.000 }
gfCNCPoint6[789] = {X 158.0338, Y 50.8306, Z -8.0000, A 0.000, B 0.000, C 0.000 }
gfCNCPoint6[790] = {X 159.2980, Y 50.7200, Z -8.0000, A 0.000, B 0.000, C 0.000 }
gfCNCPoint6[791] = {X 178.5335, Y 50.7200, Z -8.0000, A 0.000, B 0.000, C 0.000 }
gfCNCPoint6[792] = {X 179.7878, Y 50.8289, Z -8.0000, A 0.000, B 0.000, C 0.000 }
gfCNCPoint6[793] = {X 181.0046, Y 51.1522, Z -8.0000, A 0.000, B 0.000, C 0.000 }
gfCNCPoint6[794] = {X 182.1475, Y 51.6804, Z -8.0000, A 0.000, B 0.000, C 0.000 }
gfCNCPoint6[795] = {X 183.1823, Y 52.3976, Z -8.0000, A 0.000, B 0.000, C 0.000 }
gfCNCPoint6[796] = {X 184.0897, Y 53.2961, Z -8.0000, A 0.000, B 0.000, C 0.000 }
gfCNCPoint6[797] = {X 184.8261, Y 54.3392, Z -8.0000, A 0.000, B 0.000, C 0.000 }
gfCNCPoint6[798] = {X 185.3690, Y 55.4951, Z -8.0000, A 0.000, B 0.000, C 0.000 }
gfCNCPoint6[799] = {X 185.7015, Y 56.7280, Z -8.0000, A 0.000, B 0.000, C 0.000 }
gfCNCPoint6[800] = {X 185.8135, Y 58.0000, Z -8.0000, A 0.000, B 0.000, C 0.000 }
gfCNCPoint6[801] = {X 185.8133, Y 58.9942, Z -8.0000, A 0.000, B 0.000, C 0.000 }
gfCNCPoint6[802] = {X 185.7648, Y 59.7744, Z -8.0000, A 0.000, B 0.000, C 0.000 }
gfCNCPoint6[803] = {X 185.6330, Y 60.5449, Z -8.0000, A 0.000, B 0.000, C 0.000 }
gfCNCPoint6[804] = {X 211.4768, Y 88.7574, Z -8.0000, A 0.000, B 0.000, C 0.000 }
gfCNCPoint6[805] = {X 211.9382, Y 89.2398, Z -8.0000, A 0.000, B 0.000, C 0.000 }
gfCNCPoint6[806] = {X 212.4199, Y 89.7019, Z -8.0000, A 0.000, B 0.000, C 0.000 }
gfCNCPoint6[807] = {X 212.5965, Y 89.7389, Z -8.0000, A 0.000, B 0.000, C 0.000 }
gfCNCPoint6[808] = {X 213.4333, Y 89.8443, Z -8.0000, A 0.000, B 0.000, C 0.000 }
gfCNCPoint6[809] = {X 214.4204, Y 89.7706, Z -8.0000, A 0.000, B 0.000, C 0.000 }
gfCNCPoint6[810] = {X 215.4086, Y 89.7156, Z -8.0000, A 0.000, B 0.000, C 0.000 }
gfCNCPoint6[811] = {X 215.6229, Y 89.6935, Z -8.0000, A 0.000, B 0.000, C 0.000 }
gfCNCPoint6[812] = {X 215.8199, Y 89.6062, Z -8.0000, A 0.000, B 0.000, C 0.000 }
gfCNCPoint6[813] = {X 239.3446, Y 74.5358, Z -8.0000, A 0.000, B 0.000, C 0.000 }
gfCNCPoint6[814] = {X 220.5440, Y 67.1584, Z -8.0000, A 0.000, B 0.000, C 0.000 }
gfCNCPoint6[815] = {X 219.0947, Y 66.6722, Z -8.0000, A 0.000, B 0.000, C 0.000 }
gfCNCPoint6[816] = {X 217.5994, Y 66.3545, Z -8.0000, A 0.000, B 0.000, C 0.000 }
gfCNCPoint6[817] = {X 216.0776, Y 66.2097, Z -8.0000, A 0.000, B 0.000, C 0.000 }
gfCNCPoint6[818] = {X 214.8511, Y 66.0621, Z -8.0000, A 0.000, B 0.000, C 0.000 }
gfCNCPoint6[819] = {X 213.6672, Y 65.7093, Z -8.0000, A 0.000, B 0.000, C 0.000 }
gfCNCPoint6[820] = {X 212.5600, Y 65.1614, Z -8.0000, A 0.000, B 0.000, C 0.000 }
gfCNCPoint6[821] = {X 211.5613, Y 64.4341, Z -8.0000, A 0.000, B 0.000, C 0.000 }
gfCNCPoint6[822] = {X 210.7000, Y 63.5485, Z -8.0000, A 0.000, B 0.000, C 0.000 }
gfCNCPoint6[823] = {X 210.0009, Y 62.5300, Z -8.0000, A 0.000, B 0.000, C 0.000 }
gfCNCPoint6[824] = {X 209.4840, Y 61.4079, Z -8.0000, A 0.000, B 0.000, C 0.000 }
gfCNCPoint6[825] = {X 209.1643, Y 60.2146, Z -8.0000, A 0.000, B 0.000, C 0.000 }
gfCNCPoint6[826] = {X 209.0510, Y 58.9845, Z -8.0000, A 0.000, B 0.000, C 0.000 }
gfCNCPoint6[827] = {X 209.0508, Y 58.0000, Z -8.0000, A 0.000, B 0.000, C 0.000 }
gfCNCPoint6[828] = {X 209.1477, Y 56.8162, Z -8.0000, A 0.000, B 0.000, C 0.000 }
gfCNCPoint6[829] = {X 209.4358, Y 55.6638, Z -8.0000, A 0.000, B 0.000, C 0.000 }
gfCNCPoint6[830] = {X 209.9075, Y 54.5737, Z -8.0000, A 0.000, B 0.000, C 0.000 }
gfCNCPoint6[831] = {X 210.5502, Y 53.5748, Z -8.0000, A 0.000, B 0.000, C 0.000 }
gfCNCPoint6[832] = {X 211.3467, Y 52.6937, Z -8.0000, A 0.000, B 0.000, C 0.000 }
gfCNCPoint6[833] = {X 212.2759, Y 51.9538, Z -8.0000, A 0.000, B 0.000, C 0.000 }
gfCNCPoint6[834] = {X 213.3131, Y 51.3749, Z -8.0000, A 0.000, B 0.000, C 0.000 }
gfCNCPoint6[835] = {X 214.4306, Y 50.9724, Z -8.0000, A 0.000, B 0.000, C 0.000 }
gfCNCPoint6[836] = {X 215.3724, Y 50.7834, Z -8.0000, A 0.000, B 0.000, C 0.000 }
gfCNCPoint6[837] = {X 216.3308, Y 50.7200, Z -8.0000, A 0.000, B 0.000, C 0.000 }
gfCNCPoint6[838] = {X 237.2617, Y 50.7200, Z -8.0000, A 0.000, B 0.000, C 0.000 }
gfCNCPoint6[839] = {X 238.3057, Y 50.7953, Z -8.0000, A 0.000, B 0.000, C 0.000 }
gfCNCPoint6[840] = {X 239.3282, Y 51.0195, Z -8.0000, A 0.000, B 0.000, C 0.000 }
gfCNCPoint6[841] = {X 240.3080, Y 51.3880, Z -8.0000, A 0.000, B 0.000, C 0.000 }
gfCNCPoint6[842] = {X 241.2247, Y 51.8932, Z -8.0000, A 0.000, B 0.000, C 0.000 }
gfCNCPoint6[843] = {X 242.0740, Y 52.5374, Z -8.0000, A 0.000, B 0.000, C 0.000 }
gfCNCPoint6[844] = {X 242.8201, Y 53.2987, Z -8.0000, A 0.000, B 0.000, C 0.000 }
gfCNCPoint6[845] = {X 243.4470, Y 54.1607, Z -8.0000, A 0.000, B 0.000, C 0.000 }
gfCNCPoint6[846] = {X 243.9414, Y 55.1051, Z -8.0000, A 0.000, B 0.000, C 0.000 }
gfCNCPoint6[847] = {X 244.2925, Y 56.1115, Z -8.0000, A 0.000, B 0.000, C 0.000 }
gfCNCPoint6[848] = {X 249.2046, Y 58.0271, Z -8.0000, A 0.000, B 0.000, C 0.000 }
gfCNCPoint6[849] = {X 272.6714, Y 67.3415, Z -8.0000, A 0.000, B 0.000, C 0.000 }
gfCNCPoint6[850] = {X 272.6713, Y 65.2835, Z -8.0000, A 0.000, B 0.000, C 0.000 }
gfCNCPoint6[851] = {X 271.6641, Y 64.6021, Z -8.0000, A 0.000, B 0.000, C 0.000 }
gfCNCPoint6[852] = {X 270.7843, Y 63.7625, Z -8.0000, A 0.000, B 0.000, C 0.000 }
gfCNCPoint6[853] = {X 270.0566, Y 62.7882, Z -8.0000, A 0.000, B 0.000, C 0.000 }
gfCNCPoint6[854] = {X 269.5012, Y 61.7063, Z -8.0000, A 0.000, B 0.000, C 0.000 }
gfCNCPoint6[855] = {X 269.2025, Y 60.8249, Z -8.0000, A 0.000, B 0.000, C 0.000 }
gfCNCPoint6[856] = {X 269.0188, Y 59.9127, Z -8.0000, A 0.000, B 0.000, C 0.000 }
gfCNCPoint6[857] = {X 268.9529, Y 58.9845, Z -8.0000, A 0.000, B 0.000, C 0.000 }
gfCNCPoint6[858] = {X 268.9527, Y 58.0000, Z -8.0000, A 0.000, B 0.000, C 0.000 }
gfCNCPoint6[859] = {X 269.0633, Y 56.7358, Z -8.0000, A 0.000, B 0.000, C 0.000 }
gfCNCPoint6[860] = {X 269.3917, Y 55.5101, Z -8.0000, A 0.000, B 0.000, C 0.000 }
gfCNCPoint6[861] = {X 269.9280, Y 54.3600, Z -8.0000, A 0.000, B 0.000, C 0.000 }
gfCNCPoint6[862] = {X 270.6559, Y 53.3205, Z -8.0000, A 0.000, B 0.000, C 0.000 }
gfCNCPoint6[863] = {X 271.5532, Y 52.4232, Z -8.0000, A 0.000, B 0.000, C 0.000 }
gfCNCPoint6[864] = {X 272.5927, Y 51.6953, Z -8.0000, A 0.000, B 0.000, C 0.000 }
gfCNCPoint6[865] = {X 273.7428, Y 51.1590, Z -8.0000, A 0.000, B 0.000, C 0.000 }
gfCNCPoint6[866] = {X 274.9685, Y 50.8306, Z -8.0000, A 0.000, B 0.000, C 0.000 }
gfCNCPoint6[867] = {X 276.2327, Y 50.7200, Z -8.0000, A 0.000, B 0.000, C 0.000 }
gfCNCPoint6[868] = {X 292.7731, Y 50.7200, Z -8.0000, A 0.000, B 0.000, C 0.000 }
gfCNCPoint6[869] = {X 293.4209, Y 50.7489, Z -8.0000, A 0.000, B 0.000, C 0.000 }
gfCNCPoint6[870] = {X 294.0636, Y 50.8353, Z -8.0000, A 0.000, B 0.000, C 0.000 }
gfCNCPoint6[871] = {X 294.7292, Y 50.9877, Z -8.0000, A 0.000, B 0.000, C 0.000 }
gfCNCPoint6[872] = {X 295.3775, Y 51.2018, Z -8.0000, A 0.000, B 0.000, C 0.000 }
gfCNCPoint6[873] = {X 298.3089, Y 43.5503, Z -8.0000, A 0.000, B 0.000, C 0.000 }
gfCNCPoint6[874] = {X 298.4820, Y 42.5277, Z -8.0000, A 0.000, B 0.000, C 0.000 }
gfCNCPoint6[875] = {X 298.7922, Y 41.5381, Z -8.0000, A 0.000, B 0.000, C 0.000 }
gfCNCPoint6[876] = {X 299.2337, Y 40.5997, Z -8.0000, A 0.000, B 0.000, C 0.000 }
gfCNCPoint6[877] = {X 299.7984, Y 39.7298, Z -8.0000, A 0.000, B 0.000, C 0.000 }
gfCNCPoint6[878] = {X 299.7984, Y 36.9943, Z -8.0000, A 0.000, B 0.000, C 0.000 }
gfCNCPoint6[879] = {X 296.8152, Y 36.9943, Z -8.0000, A 0.000, B 0.000, C 0.000 }
gfCNCPoint6[880] = {X 296.8150, Y 39.7478, Z -8.0000, A 0.000, B 0.000, C 0.000 }
gfCNCPoint6[881] = {X 297.3859, Y 40.6100, Z -8.0000, A 0.000, B 0.000, C 0.000 }
gfCNCPoint6[882] = {X 297.8306, Y 41.5435, Z -8.0000, A 0.000, B 0.000, C 0.000 }
gfCNCPoint6[883] = {X 298.1403, Y 42.5301, Z -8.0000, A 0.000, B 0.000, C 0.000 }
gfCNCPoint6[884] = {X 298.3089, Y 43.5503, Z -8.0000, A 0.000, B 0.000, C 0.000 }
gfCNCPoint6[885] = {X 296.2362, Y 48.9607, Z -8.0000, A 0.000, B 0.000, C 0.000 }
gfCNCPoint6[886] = {X 296.6123, Y 49.1139, Z -8.0000, A 0.000, B 0.000, C 0.000 }
gfCNCPoint6[887] = {X 296.9817, Y 49.2828, Z -8.0000, A 0.000, B 0.000, C 0.000 }
gfCNCPoint6[888] = {X 297.2571, Y 49.4212, Z -8.0000, A 0.000, B 0.000, C 0.000 }
gfCNCPoint6[889] = {X 297.5280, Y 49.5683, Z -8.0000, A 0.000, B 0.000, C 0.000 }
gfCNCPoint6[890] = {X 298.7174, Y 50.3602, Z -8.0000, A 0.000, B 0.000, C 0.000 }
gfCNCPoint6[891] = {X 299.7774, Y 51.3185, Z -8.0000, A 0.000, B 0.000, C 0.000 }
gfCNCPoint6[892] = {X 300.6847, Y 52.4224, Z -8.0000, A 0.000, B 0.000, C 0.000 }
gfCNCPoint6[893] = {X 301.5914, Y 51.3191, Z -8.0000, A 0.000, B 0.000, C 0.000 }
gfCNCPoint6[894] = {X 302.6506, Y 50.3611, Z -8.0000, A 0.000, B 0.000, C 0.000 }
gfCNCPoint6[895] = {X 303.8393, Y 49.5695, Z -8.0000, A 0.000, B 0.000, C 0.000 }
gfCNCPoint6[896] = {X 302.8989, Y 49.0956, Z -8.0000, A 0.000, B 0.000, C 0.000 }
gfCNCPoint6[897] = {X 302.0820, Y 48.4310, Z -8.0000, A 0.000, B 0.000, C 0.000 }
gfCNCPoint6[898] = {X 301.4268, Y 47.6067, Z -8.0000, A 0.000, B 0.000, C 0.000 }
gfCNCPoint6[899] = {X 300.9636, Y 46.6610, Z -8.0000, A 0.000, B 0.000, C 0.000 }
gfCNCPoint6[900] = {X 300.7923, Y 46.0759, Z -8.0000, A 0.000, B 0.000, C 0.000 }
gfCNCPoint6[901] = {X 300.6953, Y 45.4741, Z -8.0000, A 0.000, B 0.000, C 0.000 }
gfCNCPoint6[902] = {X 300.6790, Y 45.2570, Z -8.0000, A 0.000, B 0.000, C 0.000 }
gfCNCPoint6[903] = {X 300.6724, Y 45.0393, Z -8.0000, A 0.000, B 0.000, C 0.000 }
gfCNCPoint6[904] = {X 300.6725, Y 44.1885, Z -8.0000, A 0.000, B 0.000, C 0.000 }
gfCNCPoint6[905] = {X 300.6809, Y 43.9886, Z -8.0000, A 0.000, B 0.000, C 0.000 }
gfCNCPoint6[906] = {X 300.6970, Y 43.7890, Z -8.0000, A 0.000, B 0.000, C 0.000 }
gfCNCPoint6[907] = {X 300.8616, Y 42.9105, Z -8.0000, A 0.000, B 0.000, C 0.000 }
gfCNCPoint6[908] = {X 301.1735, Y 42.0728, Z -8.0000, A 0.000, B 0.000, C 0.000 }
gfCNCPoint6[909] = {X 301.6235, Y 41.3004, Z -8.0000, A 0.000, B 0.000, C 0.000 }
gfCNCPoint6[910] = {X 302.1984, Y 40.6160, Z -8.0000, A 0.000, B 0.000, C 0.000 }
gfCNCPoint6[911] = {X 302.1984, Y 34.5943, Z -8.0000, A 0.000, B 0.000, C 0.000 }
gfCNCPoint6[912] = {X 294.4154, Y 34.5943, Z -8.0000, A 0.000, B 0.000, C 0.000 }
gfCNCPoint6[913] = {X 294.4149, Y 40.6548, Z -8.0000, A 0.000, B 0.000, C 0.000 }
gfCNCPoint6[914] = {X 294.9948, Y 41.3211, Z -8.0000, A 0.000, B 0.000, C 0.000 }
gfCNCPoint6[915] = {X 295.4476, Y 42.0795, Z -8.0000, A 0.000, B 0.000, C 0.000 }
gfCNCPoint6[916] = {X 295.7591, Y 42.9061, Z -8.0000, A 0.000, B 0.000, C 0.000 }
gfCNCPoint6[917] = {X 295.9195, Y 43.7747, Z -8.0000, A 0.000, B 0.000, C 0.000 }
gfCNCPoint6[918] = {X 295.9350, Y 43.9915, Z -8.0000, A 0.000, B 0.000, C 0.000 }
gfCNCPoint6[919] = {X 295.9411, Y 44.2089, Z -8.0000, A 0.000, B 0.000, C 0.000 }
gfCNCPoint6[920] = {X 295.9411, Y 45.0000, Z -8.0000, A 0.000, B 0.000, C 0.000 }
gfCNCPoint6[921] = {X 295.9354, Y 45.2373, Z -8.0000, A 0.000, B 0.000, C 0.000 }
gfCNCPoint6[922] = {X 295.9180, Y 45.4741, Z -8.0000, A 0.000, B 0.000, C 0.000 }
gfCNCPoint6[923] = {X 298.3067, Y 45.7073, Z -8.0000, A 0.000, B 0.000, C 0.000 }
gfCNCPoint6[924] = {X 298.2010, Y 46.4214, Z -8.0000, A 0.000, B 0.000, C 0.000 }
gfCNCPoint6[925] = {X 298.0252, Y 47.1215, Z -8.0000, A 0.000, B 0.000, C 0.000 }
gfCNCPoint6[926] = {X 298.3689, Y 47.2942, Z -8.0000, A 0.000, B 0.000, C 0.000 }
gfCNCPoint6[927] = {X 298.7069, Y 47.4778, Z -8.0000, A 0.000, B 0.000, C 0.000 }
gfCNCPoint6[928] = {X 298.4514, Y 46.6051, Z -8.0000, A 0.000, B 0.000, C 0.000 }
gfCNCPoint6[929] = {X 298.3067, Y 45.7073, Z -8.0000, A 0.000, B 0.000, C 0.000 }
gfCNCPoint6[930] = {X 295.9180, Y 45.4741, Z -8.0000, A 0.000, B 0.000, C 0.000 }
gfCNCPoint6[931] = {X 295.8472, Y 45.9528, Z -8.0000, A 0.000, B 0.000, C 0.000 }
gfCNCPoint6[932] = {X 295.7293, Y 46.4221, Z -8.0000, A 0.000, B 0.000, C 0.000 }
gfCNCPoint6[933] = {X 295.4314, Y 47.1714, Z -8.0000, A 0.000, B 0.000, C 0.000 }
gfCNCPoint6[934] = {X 295.0142, Y 47.8614, Z -8.0000, A 0.000, B 0.000, C 0.000 }
gfCNCPoint6[935] = {X 294.4890, Y 48.4733, Z -8.0000, A 0.000, B 0.000, C 0.000 }
gfCNCPoint6[936] = {X 295.3740, Y 48.6760, Z -8.0000, A 0.000, B 0.000, C 0.000 }
gfCNCPoint6[937] = {X 296.2362, Y 48.9607, Z -8.0000, A 0.000, B 0.000, C 0.000 }
gfCNCPoint6[938] = {X 295.3775, Y 51.2018, Z -8.0000, A 0.000, B 0.000, C 0.000 }
gfCNCPoint6[939] = {X 296.3497, Y 51.6592, Z -8.0000, A 0.000, B 0.000, C 0.000 }
gfCNCPoint6[940] = {X 297.2440, Y 52.2546, Z -8.0000, A 0.000, B 0.000, C 0.000 }
gfCNCPoint6[941] = {X 298.0409, Y 52.9752, Z -8.0000, A 0.000, B 0.000, C 0.000 }
gfCNCPoint6[942] = {X 298.7231, Y 53.8053, Z -8.0000, A 0.000, B 0.000, C 0.000 }
gfCNCPoint6[943] = {X 299.2946, Y 54.7645, Z -8.0000, A 0.000, B 0.000, C 0.000 }
gfCNCPoint6[944] = {X 299.7126, Y 55.7997, Z -8.0000, A 0.000, B 0.000, C 0.000 }
gfCNCPoint6[945] = {X 299.9675, Y 56.8868, Z -8.0000, A 0.000, B 0.000, C 0.000 }
gfCNCPoint6[946] = {X 300.0531, Y 58.0000, Z -8.0000, A 0.000, B 0.000, C 0.000 }
gfCNCPoint6[947] = {X 300.0531, Y 58.9428, Z -8.0000, A 0.000, B 0.000, C 0.000 }
gfCNCPoint6[948] = {X 299.9651, Y 60.0531, Z -8.0000, A 0.000, B 0.000, C 0.000 }
gfCNCPoint6[949] = {X 299.7092, Y 61.1372, Z -8.0000, A 0.000, B 0.000, C 0.000 }
gfCNCPoint6[950] = {X 299.2912, Y 62.1696, Z -8.0000, A 0.000, B 0.000, C 0.000 }
gfCNCPoint6[951] = {X 298.7209, Y 63.1263, Z -8.0000, A 0.000, B 0.000, C 0.000 }
gfCNCPoint6[952] = {X 300.6827, Y 64.5089, Z -8.0000, A 0.000, B 0.000, C 0.000 }
gfCNCPoint6[953] = {X 299.7835, Y 65.6049, Z -8.0000, A 0.000, B 0.000, C 0.000 }
gfCNCPoint6[954] = {X 298.7341, Y 66.5581, Z -8.0000, A 0.000, B 0.000, C 0.000 }
gfCNCPoint6[955] = {X 298.7341, Y 89.4416, Z -8.0000, A 0.000, B 0.000, C 0.000 }
gfCNCPoint6[956] = {X 299.8307, Y 90.4462, Z -8.0000, A 0.000, B 0.000, C 0.000 }
gfCNCPoint6[957] = {X 300.7610, Y 91.6065, Z -8.0000, A 0.000, B 0.000, C 0.000 }
gfCNCPoint6[958] = {X 301.5033, Y 92.8952, Z -8.0000, A 0.000, B 0.000, C 0.000 }
gfCNCPoint6[959] = {X 304.0681, Y 92.8952, Z -8.0000, A 0.000, B 0.000, C 0.000 }
gfCNCPoint6[960] = {X 303.4736, Y 91.0762, Z -8.0000, A 0.000, B 0.000, C 0.000 }
gfCNCPoint6[961] = {X 303.0368, Y 89.2129, Z -8.0000, A 0.000, B 0.000, C 0.000 }
gfCNCPoint6[962] = {X 302.7611, Y 87.3192, Z -8.0000, A 0.000, B 0.000, C 0.000 }
gfCNCPoint6[963] = {X 302.6485, Y 85.4088, Z -8.0000, A 0.000, B 0.000, C 0.000 }
gfCNCPoint6[964] = {X 302.6340, Y 84.6391, Z -8.0000, A 0.000, B 0.000, C 0.000 }
gfCNCPoint6[965] = {X 302.6351, Y 66.5608, Z -8.0000, A 0.000, B 0.000, C 0.000 }
gfCNCPoint6[966] = {X 301.5834, Y 65.6066, Z -8.0000, A 0.000, B 0.000, C 0.000 }
gfCNCPoint6[967] = {X 300.6827, Y 64.5089, Z -8.0000, A 0.000, B 0.000, C 0.000 }
gfCNCPoint6[968] = {X 298.7209, Y 63.1263, Z -8.0000, A 0.000, B 0.000, C 0.000 }
gfCNCPoint6[969] = {X 298.0351, Y 63.9607, Z -8.0000, A 0.000, B 0.000, C 0.000 }
gfCNCPoint6[970] = {X 297.2337, Y 64.6847, Z -8.0000, A 0.000, B 0.000, C 0.000 }
gfCNCPoint6[971] = {X 296.3341, Y 65.2824, Z -8.0000, A 0.000, B 0.000, C 0.000 }
gfCNCPoint6[972] = {X 296.3341, Y 90.7157, Z -8.0000, A 0.000, B 0.000, C 0.000 }
gfCNCPoint6[973] = {X 297.3142, Y 91.3786, Z -8.0000, A 0.000, B 0.000, C 0.000 }
gfCNCPoint6[974] = {X 298.1745, Y 92.1908, Z -8.0000, A 0.000, B 0.000, C 0.000 }
gfCNCPoint6[975] = {X 298.8925, Y 93.1312, Z -8.0000, A 0.000, B 0.000, C 0.000 }
gfCNCPoint6[976] = {X 299.4495, Y 94.1751, Z -8.0000, A 0.000, B 0.000, C 0.000 }
gfCNCPoint6[977] = {X 299.8309, Y 95.2952, Z -8.0000, A 0.000, B 0.000, C 0.000 }
gfCNCPoint6[978] = {X 308.1032, Y 95.2952, Z -8.0000, A 0.000, B 0.000, C 0.000 }
gfCNCPoint6[979] = {X 307.1083, Y 93.7244, Z -8.0000, A 0.000, B 0.000, C 0.000 }
gfCNCPoint6[980] = {X 306.3122, Y 92.0442, Z -8.0000, A 0.000, B 0.000, C 0.000 }
gfCNCPoint6[981] = {X 305.7825, Y 90.4214, Z -8.0000, A 0.000, B 0.000, C 0.000 }
gfCNCPoint6[982] = {X 305.3936, Y 88.7594, Z -8.0000, A 0.000, B 0.000, C 0.000 }
gfCNCPoint6[983] = {X 305.1482, Y 87.0702, Z -8.0000, A 0.000, B 0.000, C 0.000 }
gfCNCPoint6[984] = {X 305.0481, Y 85.3661, Z -8.0000, A 0.000, B 0.000, C 0.000 }
gfCNCPoint6[985] = {X 305.0340, Y 84.6275, Z -8.0000, A 0.000, B 0.000, C 0.000 }
gfCNCPoint6[986] = {X 305.0352, Y 65.2837, Z -8.0000, A 0.000, B 0.000, C 0.000 }
gfCNCPoint6[987] = {X 304.1340, Y 64.6862, Z -8.0000, A 0.000, B 0.000, C 0.000 }
gfCNCPoint6[988] = {X 303.3313, Y 63.9619, Z -8.0000, A 0.000, B 0.000, C 0.000 }
gfCNCPoint6[989] = {X 302.6447, Y 63.1267, Z -8.0000, A 0.000, B 0.000, C 0.000 }
gfCNCPoint6[990] = {X 302.0795, Y 62.1792, Z -8.0000, A 0.000, B 0.000, C 0.000 }
gfCNCPoint6[991] = {X 301.6639, Y 61.1571, Z -8.0000, A 0.000, B 0.000, C 0.000 }
gfCNCPoint6[992] = {X 301.4076, Y 60.0840, Z -8.0000, A 0.000, B 0.000, C 0.000 }
gfCNCPoint6[993] = {X 301.3164, Y 58.9845, Z -8.0000, A 0.000, B 0.000, C 0.000 }
gfCNCPoint6[994] = {X 301.3162, Y 58.0000, Z -8.0000, A 0.000, B 0.000, C 0.000 }
gfCNCPoint6[995] = {X 301.4018, Y 56.8868, Z -8.0000, A 0.000, B 0.000, C 0.000 }
gfCNCPoint6[996] = {X 301.6567, Y 55.7997, Z -8.0000, A 0.000, B 0.000, C 0.000 }
gfCNCPoint6[997] = {X 302.0747, Y 54.7645, Z -8.0000, A 0.000, B 0.000, C 0.000 }
gfCNCPoint6[998] = {X 302.6462, Y 53.8053, Z -8.0000, A 0.000, B 0.000, C 0.000 }
gfCNCPoint6[999] = {X 303.3281, Y 52.9755, Z -8.0000, A 0.000, B 0.000, C 0.000 }
gfCNCPoint6[1000] = {X 304.1247, Y 52.2551, Z -8.0000, A 0.000, B 0.000, C 0.000 }
gfCNCPoint6[1001] = {X 305.0187, Y 51.6597, Z -8.0000, A 0.000, B 0.000, C 0.000 }
gfCNCPoint6[1002] = {X 306.1514, Y 51.1428, Z -8.0000, A 0.000, B 0.000, C 0.000 }
gfCNCPoint6[1003] = {X 307.3557, Y 50.8265, Z -8.0000, A 0.000, B 0.000, C 0.000 }
gfCNCPoint6[1004] = {X 308.5962, Y 50.7200, Z -8.0000, A 0.000, B 0.000, C 0.000 }
gfCNCPoint6[1005] = {X 324.3107, Y 50.7200, Z -8.0000, A 0.000, B 0.000, C 0.000 }
gfCNCPoint6[1006] = {X 325.2469, Y 50.7804, Z -8.0000, A 0.000, B 0.000, C 0.000 }
gfCNCPoint6[1007] = {X 326.1675, Y 50.9608, Z -8.0000, A 0.000, B 0.000, C 0.000 }
gfCNCPoint6[1008] = {X 326.5260, Y 51.0653, Z -8.0000, A 0.000, B 0.000, C 0.000 }
gfCNCPoint6[1009] = {X 326.8787, Y 51.1880, Z -8.0000, A 0.000, B 0.000, C 0.000 }
gfCNCPoint6[1010] = {X 327.4496, Y 51.4315, Z -8.0000, A 0.000, B 0.000, C 0.000 }
gfCNCPoint6[1011] = {X 327.9977, Y 51.7227, Z -8.0000, A 0.000, B 0.000, C 0.000 }
gfCNCPoint6[1012] = {X 328.5432, Y 52.0768, Z -8.0000, A 0.000, B 0.000, C 0.000 }
gfCNCPoint6[1013] = {X 329.0549, Y 52.4782, Z -8.0000, A 0.000, B 0.000, C 0.000 }
gfCNCPoint6[1014] = {X 329.9309, Y 53.3727, Z -8.0000, A 0.000, B 0.000, C 0.000 }
gfCNCPoint6[1015] = {X 330.6407, Y 54.4042, Z -8.0000, A 0.000, B 0.000, C 0.000 }
gfCNCPoint6[1016] = {X 331.1632, Y 55.5420, Z -8.0000, A 0.000, B 0.000, C 0.000 }
gfCNCPoint6[1017] = {X 331.4830, Y 56.7526, Z -8.0000, A 0.000, B 0.000, C 0.000 }
gfCNCPoint6[1018] = {X 331.5907, Y 58.0000, Z -8.0000, A 0.000, B 0.000, C 0.000 }
gfCNCPoint6[1019] = {X 331.5907, Y 58.9391, Z -8.0000, A 0.000, B 0.000, C 0.000 }
gfCNCPoint6[1020] = {X 331.4738, Y 60.2163, Z -8.0000, A 0.000, B 0.000, C 0.000 }
gfCNCPoint6[1021] = {X 331.1357, Y 61.4535, Z -8.0000, A 0.000, B 0.000, C 0.000 }
gfCNCPoint6[1022] = {X 330.5868, Y 62.6126, Z -8.0000, A 0.000, B 0.000, C 0.000 }
gfCNCPoint6[1023] = {X 329.8439, Y 63.6580, Z -8.0000, A 0.000, B 0.000, C 0.000 }
gfCNCPoint6[1024] = {X 328.9299, Y 64.5577, Z -8.0000, A 0.000, B 0.000, C 0.000 }
gfCNCPoint6[1025] = {X 327.8728, Y 65.2840, Z -8.0000, A 0.000, B 0.000, C 0.000 }
gfCNCPoint6[1026] = {X 327.8746, Y 83.2150, Z -8.0000, A 0.000, B 0.000, C 0.000 }
gfCNCPoint6[1027] = {X 327.8880, Y 84.5909, Z -8.0000, A 0.000, B 0.000, C 0.000 }
gfCNCPoint6[1028] = {X 327.8976, Y 84.9517, Z -8.0000, A 0.000, B 0.000, C 0.000 }
gfCNCPoint6[1029] = {X 327.9242, Y 85.3117, Z -8.0000, A 0.000, B 0.000, C 0.000 }
gfCNCPoint6[1030] = {X 329.1613, Y 85.7649, Z -8.0000, A 0.000, B 0.000, C 0.000 }
gfCNCPoint6[1031] = {X 330.4379, Y 86.0906, Z -8.0000, A 0.000, B 0.000, C 0.000 }
gfCNCPoint6[1032] = {X 333.3491, Y 86.6136, Z -8.0000, A 0.000, B 0.000, C 0.000 }
gfCNCPoint6[1033] = {X 336.2867, Y 86.9580, Z -8.0000, A 0.000, B 0.000, C 0.000 }
gfCNCPoint6[1034] = {X 340.5661, Y 87.2459, Z -8.0000, A 0.000, B 0.000, C 0.000 }
gfCNCPoint6[1035] = {X 344.8524, Y 87.3962, Z -8.0000, A 0.000, B 0.000, C 0.000 }
gfCNCPoint6[1036] = {X 349.1414, Y 87.4087, Z -8.0000, A 0.000, B 0.000, C 0.000 }
gfCNCPoint6[1037] = {X 353.1932, Y 87.3428, Z -8.0000, A 0.000, B 0.000, C 0.000 }
gfCNCPoint6[1038] = {X 357.2399, Y 87.1296, Z -8.0000, A 0.000, B 0.000, C 0.000 }
gfCNCPoint6[1039] = {X 361.2762, Y 86.7694, Z -8.0000, A 0.000, B 0.000, C 0.000 }
gfCNCPoint6[1040] = {X 363.1974, Y 86.5041, Z -8.0000, A 0.000, B 0.000, C 0.000 }
gfCNCPoint6[1041] = {X 365.1008, Y 86.1327, Z -8.0000, A 0.000, B 0.000, C 0.000 }
gfCNCPoint6[1042] = {X 366.9808, Y 85.6562, Z -8.0000, A 0.000, B 0.000, C 0.000 }
gfCNCPoint6[1043] = {X 367.4411, Y 85.5103, Z -8.0000, A 0.000, B 0.000, C 0.000 }
gfCNCPoint6[1044] = {X 367.8876, Y 85.3263, Z -8.0000, A 0.000, B 0.000, C 0.000 }
gfCNCPoint6[1045] = {X 367.9410, Y 84.5786, Z -8.0000, A 0.000, B 0.000, C 0.000 }
gfCNCPoint6[1046] = {X 367.9587, Y 83.8292, Z -8.0000, A 0.000, B 0.000, C 0.000 }
gfCNCPoint6[1047] = {X 367.9577, Y 65.2834, Z -8.0000, A 0.000, B 0.000, C 0.000 }
gfCNCPoint6[1048] = {X 366.9042, Y 64.5643, Z -8.0000, A 0.000, B 0.000, C 0.000 }
gfCNCPoint6[1049] = {X 365.9923, Y 63.6723, Z -8.0000, A 0.000, B 0.000, C 0.000 }
gfCNCPoint6[1050] = {X 365.2501, Y 62.6348, Z -8.0000, A 0.000, B 0.000, C 0.000 }
gfCNCPoint6[1051] = {X 364.7004, Y 61.4837, Z -8.0000, A 0.000, B 0.000, C 0.000 }
gfCNCPoint6[1052] = {X 364.3600, Y 60.2544, Z -8.0000, A 0.000, B 0.000, C 0.000 }
gfCNCPoint6[1053] = {X 364.2395, Y 58.9845, Z -8.0000, A 0.000, B 0.000, C 0.000 }
gfCNCPoint6[1054] = {X 364.2393, Y 58.0000, Z -8.0000, A 0.000, B 0.000, C 0.000 }
gfCNCPoint6[1055] = {X 364.3499, Y 56.7358, Z -8.0000, A 0.000, B 0.000, C 0.000 }
gfCNCPoint6[1056] = {X 364.6783, Y 55.5101, Z -8.0000, A 0.000, B 0.000, C 0.000 }
gfCNCPoint6[1057] = {X 365.2146, Y 54.3600, Z -8.0000, A 0.000, B 0.000, C 0.000 }
gfCNCPoint6[1058] = {X 365.9425, Y 53.3205, Z -8.0000, A 0.000, B 0.000, C 0.000 }
gfCNCPoint6[1059] = {X 366.8398, Y 52.4232, Z -8.0000, A 0.000, B 0.000, C 0.000 }
gfCNCPoint6[1060] = {X 367.8793, Y 51.6953, Z -8.0000, A 0.000, B 0.000, C 0.000 }
gfCNCPoint6[1061] = {X 369.0294, Y 51.1590, Z -8.0000, A 0.000, B 0.000, C 0.000 }
gfCNCPoint6[1062] = {X 370.2551, Y 50.8306, Z -8.0000, A 0.000, B 0.000, C 0.000 }
gfCNCPoint6[1063] = {X 371.5193, Y 50.7200, Z -8.0000, A 0.000, B 0.000, C 0.000 }
gfCNCPoint6[1064] = {X 388.0597, Y 50.7200, Z -8.0000, A 0.000, B 0.000, C 0.000 }
gfCNCPoint6[1065] = {X 389.2271, Y 50.8142, Z -8.0000, A 0.000, B 0.000, C 0.000 }
gfCNCPoint6[1066] = {X 390.3643, Y 51.0944, Z -8.0000, A 0.000, B 0.000, C 0.000 }
gfCNCPoint6[1067] = {X 391.4418, Y 51.5533, Z -8.0000, A 0.000, B 0.000, C 0.000 }
gfCNCPoint6[1068] = {X 392.4319, Y 52.1791, Z -8.0000, A 0.000, B 0.000, C 0.000 }
gfCNCPoint6[1069] = {X 393.3087, Y 52.9556, Z -8.0000, A 0.000, B 0.000, C 0.000 }
gfCNCPoint6[1070] = {X 394.1855, Y 52.1791, Z -8.0000, A 0.000, B 0.000, C 0.000 }
gfCNCPoint6[1071] = {X 395.1756, Y 51.5533, Z -8.0000, A 0.000, B 0.000, C 0.000 }
gfCNCPoint6[1072] = {X 396.2531, Y 51.0944, Z -8.0000, A 0.000, B 0.000, C 0.000 }
gfCNCPoint6[1073] = {X 397.3903, Y 50.8142, Z -8.0000, A 0.000, B 0.000, C 0.000 }
gfCNCPoint6[1074] = {X 398.5577, Y 50.7200, Z -8.0000, A 0.000, B 0.000, C 0.000 }
gfCNCPoint6[1075] = {X 419.4886, Y 50.7200, Z -8.0000, A 0.000, B 0.000, C 0.000 }
gfCNCPoint6[1076] = {X 420.6738, Y 50.8171, Z -8.0000, A 0.000, B 0.000, C 0.000 }
gfCNCPoint6[1077] = {X 421.8274, Y 51.1059, Z -8.0000, A 0.000, B 0.000, C 0.000 }
gfCNCPoint6[1078] = {X 422.9186, Y 51.5787, Z -8.0000, A 0.000, B 0.000, C 0.000 }
gfCNCPoint6[1079] = {X 423.9183, Y 52.2228, Z -8.0000, A 0.000, B 0.000, C 0.000 }
gfCNCPoint6[1080] = {X 424.7997, Y 53.0210, Z -8.0000, A 0.000, B 0.000, C 0.000 }
gfCNCPoint6[1081] = {X 425.5395, Y 53.9521, Z -8.0000, A 0.000, B 0.000, C 0.000 }
gfCNCPoint6[1082] = {X 426.1178, Y 54.9912, Z -8.0000, A 0.000, B 0.000, C 0.000 }
gfCNCPoint6[1083] = {X 426.5192, Y 56.1106, Z -8.0000, A 0.000, B 0.000, C 0.000 }
gfCNCPoint6[1084] = {X 430.7007, Y 57.7397, Z -8.0000, A 0.000, B 0.000, C 0.000 }
gfCNCPoint6[1085] = {X 454.8979, Y 67.3406, Z -8.0000, A 0.000, B 0.000, C 0.000 }
gfCNCPoint6[1086] = {X 454.8980, Y 65.2833, Z -8.0000, A 0.000, B 0.000, C 0.000 }
gfCNCPoint6[1087] = {X 453.8908, Y 64.6019, Z -8.0000, A 0.000, B 0.000, C 0.000 }
gfCNCPoint6[1088] = {X 453.0112, Y 63.7624, Z -8.0000, A 0.000, B 0.000, C 0.000 }
gfCNCPoint6[1089] = {X 452.2835, Y 62.7882, Z -8.0000, A 0.000, B 0.000, C 0.000 }
gfCNCPoint6[1090] = {X 451.7281, Y 61.7064, Z -8.0000, A 0.000, B 0.000, C 0.000 }
gfCNCPoint6[1091] = {X 451.4295, Y 60.8250, Z -8.0000, A 0.000, B 0.000, C 0.000 }
gfCNCPoint6[1092] = {X 451.2457, Y 59.9128, Z -8.0000, A 0.000, B 0.000, C 0.000 }
gfCNCPoint6[1093] = {X 451.1798, Y 58.9845, Z -8.0000, A 0.000, B 0.000, C 0.000 }
gfCNCPoint6[1094] = {X 451.1796, Y 58.0000, Z -8.0000, A 0.000, B 0.000, C 0.000 }
gfCNCPoint6[1095] = {X 451.2795, Y 56.7981, Z -8.0000, A 0.000, B 0.000, C 0.000 }
gfCNCPoint6[1096] = {X 451.5765, Y 55.6291, Z -8.0000, A 0.000, B 0.000, C 0.000 }
gfCNCPoint6[1097] = {X 452.0624, Y 54.5253, Z -8.0000, A 0.000, B 0.000, C 0.000 }
gfCNCPoint6[1098] = {X 452.7238, Y 53.5168, Z -8.0000, A 0.000, B 0.000, C 0.000 }
gfCNCPoint6[1099] = {X 453.5427, Y 52.6313, Z -8.0000, A 0.000, B 0.000, C 0.000 }
gfCNCPoint6[1100] = {X 454.4966, Y 51.8932, Z -8.0000, A 0.000, B 0.000, C 0.000 }
gfCNCPoint6[1101] = {X 455.4133, Y 51.3880, Z -8.0000, A 0.000, B 0.000, C 0.000 }
gfCNCPoint6[1102] = {X 456.3931, Y 51.0195, Z -8.0000, A 0.000, B 0.000, C 0.000 }
gfCNCPoint6[1103] = {X 457.4155, Y 50.7953, Z -8.0000, A 0.000, B 0.000, C 0.000 }
gfCNCPoint6[1104] = {X 458.4596, Y 50.7200, Z -8.0000, A 0.000, B 0.000, C 0.000 }
gfCNCPoint6[1105] = {X 475.0000, Y 50.7200, Z -8.0000, A 0.000, B 0.000, C 0.000 }
gfCNCPoint6[1106] = {X 476.0441, Y 50.7953, Z -8.0000, A 0.000, B 0.000, C 0.000 }
gfCNCPoint6[1107] = {X 477.0665, Y 51.0195, Z -8.0000, A 0.000, B 0.000, C 0.000 }
gfCNCPoint6[1108] = {X 478.0463, Y 51.3880, Z -8.0000, A 0.000, B 0.000, C 0.000 }
gfCNCPoint6[1109] = {X 478.9630, Y 51.8932, Z -8.0000, A 0.000, B 0.000, C 0.000 }
gfCNCPoint6[1110] = {X 479.9169, Y 52.6313, Z -8.0000, A 0.000, B 0.000, C 0.000 }
gfCNCPoint6[1111] = {X 480.7358, Y 53.5168, Z -8.0000, A 0.000, B 0.000, C 0.000 }
gfCNCPoint6[1112] = {X 481.3972, Y 54.5253, Z -8.0000, A 0.000, B 0.000, C 0.000 }
gfCNCPoint6[1113] = {X 481.8831, Y 55.6291, Z -8.0000, A 0.000, B 0.000, C 0.000 }
gfCNCPoint6[1114] = {X 482.1801, Y 56.7981, Z -8.0000, A 0.000, B 0.000, C 0.000 }
gfCNCPoint6[1115] = {X 482.2800, Y 58.0000, Z -8.0000, A 0.000, B 0.000, C 0.000 }
gfCNCPoint6[1116] = {X 482.2798, Y 58.9942, Z -8.0000, A 0.000, B 0.000, C 0.000 }
gfCNCPoint6[1117] = {X 482.1578, Y 60.2624, Z -8.0000, A 0.000, B 0.000, C 0.000 }
gfCNCPoint6[1118] = {X 481.8166, Y 61.4899, Z -8.0000, A 0.000, B 0.000, C 0.000 }
gfCNCPoint6[1119] = {X 481.2666, Y 62.6391, Z -8.0000, A 0.000, B 0.000, C 0.000 }
gfCNCPoint6[1120] = {X 480.5248, Y 63.6749, Z -8.0000, A 0.000, B 0.000, C 0.000 }
gfCNCPoint6[1121] = {X 479.6137, Y 64.5655, Z -8.0000, A 0.000, B 0.000, C 0.000 }
gfCNCPoint6[1122] = {X 478.5613, Y 65.2835, Z -8.0000, A 0.000, B 0.000, C 0.000 }
gfCNCPoint6[1123] = {X 478.5617, Y 90.7242, Z -8.0000, A 0.000, B 0.000, C 0.000 }
gfCNCPoint6[1124] = {X 479.5437, Y 91.3832, Z -8.0000, A 0.000, B 0.000, C 0.000 }
gfCNCPoint6[1125] = {X 480.4058, Y 92.1929, Z -8.0000, A 0.000, B 0.000, C 0.000 }
gfCNCPoint6[1126] = {X 481.1248, Y 93.1319, Z -8.0000, A 0.000, B 0.000, C 0.000 }
gfCNCPoint6[1127] = {X 481.6818, Y 94.1753, Z -8.0000, A 0.000, B 0.000, C 0.000 }
gfCNCPoint6[1128] = {X 482.0620, Y 95.2952, Z -8.0000, A 0.000, B 0.000, C 0.000 }
gfCNCPoint6[1129] = {X 507.6811, Y 95.2952, Z -8.0000, A 0.000, B 0.000, C 0.000 }
gfCNCPoint6[1130] = {X 507.6811, Y 97.6952, Z -8.0000, A 0.000, B 0.000, C 0.000 }
gfCNCPoint6[1131] = {X 597.6967, Y 97.6952, Z -8.0000, A 0.000, B 0.000, C 0.000 }
gfCNCPoint6[1132] = {X 597.6967, Y 51.8000, Z -8.0000, A 0.000, B 0.000, C 0.000 }
gfCNCPoint6[1133] = {X 593.5565, Y 51.8000, Z -8.0000, A 0.000, B 0.000, C 0.000 }
gfCNCPoint6[1134] = {X 592.3428, Y 51.6908, Z -8.0000, A 0.000, B 0.000, C 0.000 }
gfCNCPoint6[1135] = {X 591.1680, Y 51.3667, Z -8.0000, A 0.000, B 0.000, C 0.000 }
gfCNCPoint6[1136] = {X 590.0699, Y 50.8381, Z -8.0000, A 0.000, B 0.000, C 0.000 }
gfCNCPoint6[1137] = {X 589.0838, Y 50.1220, Z -8.0000, A 0.000, B 0.000, C 0.000 }
gfCNCPoint6[1138] = {X 588.4736, Y 49.5171, Z -8.0000, A 0.000, B 0.000, C 0.000 }
gfCNCPoint6[1139] = {X 587.9446, Y 48.8401, Z -8.0000, A 0.000, B 0.000, C 0.000 }
gfCNCPoint6[1140] = {X 587.5052, Y 48.1018, Z -8.0000, A 0.000, B 0.000, C 0.000 }
gfCNCPoint6[1141] = {X 587.0658, Y 48.8401, Z -8.0000, A 0.000, B 0.000, C 0.000 }
gfCNCPoint6[1142] = {X 586.5368, Y 49.5171, Z -8.0000, A 0.000, B 0.000, C 0.000 }
gfCNCPoint6[1143] = {X 585.9266, Y 50.1220, Z -8.0000, A 0.000, B 0.000, C 0.000 }
gfCNCPoint6[1144] = {X 585.1803, Y 50.6880, Z -8.0000, A 0.000, B 0.000, C 0.000 }
gfCNCPoint6[1145] = {X 584.3634, Y 51.1461, Z -8.0000, A 0.000, B 0.000, C 0.000 }
gfCNCPoint6[1146] = {X 583.3013, Y 51.5442, Z -8.0000, A 0.000, B 0.000, C 0.000 }
gfCNCPoint6[1147] = {X 582.1877, Y 51.7603, Z -8.0000, A 0.000, B 0.000, C 0.000 }
gfCNCPoint6[1148] = {X 581.0538, Y 51.7882, Z -8.0000, A 0.000, B 0.000, C 0.000 }
gfCNCPoint6[1149] = {X 579.9310, Y 51.6273, Z -8.0000, A 0.000, B 0.000, C 0.000 }
gfCNCPoint6[1150] = {X 578.8505, Y 51.2819, Z -8.0000, A 0.000, B 0.000, C 0.000 }
gfCNCPoint6[1151] = {X 577.8425, Y 50.7618, Z -8.0000, A 0.000, B 0.000, C 0.000 }
gfCNCPoint6[1152] = {X 576.9350, Y 50.0813, Z -8.0000, A 0.000, B 0.000, C 0.000 }
gfCNCPoint6[1153] = {X 576.3133, Y 49.4513, Z -8.0000, A 0.000, B 0.000, C 0.000 }
gfCNCPoint6[1154] = {X 575.7786, Y 48.7459, Z -8.0000, A 0.000, B 0.000, C 0.000 }
gfCNCPoint6[1155] = {X 575.3401, Y 47.9770, Z -8.0000, A 0.000, B 0.000, C 0.000 }
gfCNCPoint6[1156] = {X 574.9017, Y 48.7459, Z -8.0000, A 0.000, B 0.000, C 0.000 }
gfCNCPoint6[1157] = {X 574.3670, Y 49.4513, Z -8.0000, A 0.000, B 0.000, C 0.000 }
gfCNCPoint6[1158] = {X 573.7453, Y 50.0813, Z -8.0000, A 0.000, B 0.000, C 0.000 }
gfCNCPoint6[1159] = {X 572.7526, Y 50.8143, Z -8.0000, A 0.000, B 0.000, C 0.000 }
gfCNCPoint6[1160] = {X 571.6437, Y 51.3558, Z -8.0000, A 0.000, B 0.000, C 0.000 }
gfCNCPoint6[1161] = {X 570.4553, Y 51.6880, Z -8.0000, A 0.000, B 0.000, C 0.000 }
gfCNCPoint6[1162] = {X 569.2264, Y 51.8000, Z -8.0000, A 0.000, B 0.000, C 0.000 }
gfCNCPoint6[1163] = {X 562.4443, Y 51.8000, Z -8.0000, A 0.000, B 0.000, C 0.000 }
gfCNCPoint6[1164] = {X 561.2635, Y 51.6967, Z -8.0000, A 0.000, B 0.000, C 0.000 }
gfCNCPoint6[1165] = {X 560.1186, Y 51.3899, Z -8.0000, A 0.000, B 0.000, C 0.000 }
gfCNCPoint6[1166] = {X 559.0443, Y 50.8890, Z -8.0000, A 0.000, B 0.000, C 0.000 }
gfCNCPoint6[1167] = {X 558.0733, Y 50.2091, Z -8.0000, A 0.000, B 0.000, C 0.000 }
gfCNCPoint6[1168] = {X 557.2352, Y 49.3710, Z -8.0000, A 0.000, B 0.000, C 0.000 }
gfCNCPoint6[1169] = {X 556.5553, Y 48.4000, Z -8.0000, A 0.000, B 0.000, C 0.000 }
gfCNCPoint6[1170] = {X 556.0544, Y 47.3257, Z -8.0000, A 0.000, B 0.000, C 0.000 }
gfCNCPoint6[1171] = {X 555.7476, Y 46.1808, Z -8.0000, A 0.000, B 0.000, C 0.000 }
gfCNCPoint6[1172] = {X 555.6443, Y 45.0000, Z -8.0000, A 0.000, B 0.000, C 0.000 }
gfCNCPoint6[1173] = {X 555.6443, Y 44.0571, Z -8.0000, A 0.000, B 0.000, C 0.000 }
gfCNCPoint6[1174] = {X 555.7460, Y 42.9045, Z -8.0000, A 0.000, B 0.000, C 0.000 }
gfCNCPoint6[1175] = {X 556.0408, Y 41.7857, Z -8.0000, A 0.000, B 0.000, C 0.000 }
gfCNCPoint6[1176] = {X 556.5202, Y 40.7326, Z -8.0000, A 0.000, B 0.000, C 0.000 }
gfCNCPoint6[1177] = {X 557.1706, Y 39.7756, Z -8.0000, A 0.000, B 0.000, C 0.000 }
gfCNCPoint6[1178] = {X 557.1710, Y 10.2274, Z -8.0000, A 0.000, B 0.000, C 0.000 }
gfCNCPoint6[1179] = {X 556.5252, Y 9.2814, Z -8.0000, A 0.000, B 0.000, C 0.000 }
gfCNCPoint6[1180] = {X 556.0474, Y 8.2404, Z -8.0000, A 0.000, B 0.000, C 0.000 }
gfCNCPoint6[1181] = {X 555.7510, Y 7.1340, Z -8.0000, A 0.000, B 0.000, C 0.000 }
gfCNCPoint6[1182] = {X 555.6446, Y 5.9935, Z -8.0000, A 0.000, B 0.000, C 0.000 }
gfCNCPoint6[1183] = {X 555.6443, Y 5.0000, Z -8.0000, A 0.000, B 0.000, C 0.000 }
gfCNCPoint6[1184] = {X 555.6452, Y 4.8909, Z -8.0000, A 0.000, B 0.000, C 0.000 }
gfCNCPoint6[1185] = {X 555.6478, Y 4.7818, Z -8.0000, A 0.000, B 0.000, C 0.000 }
gfCNCPoint6[1186] = {X 555.8079, Y 3.5173, Z -8.0000, A 0.000, B 0.000, C 0.000 }
gfCNCPoint6[1187] = {X 556.2012, Y 2.3048, Z -8.0000, A 0.000, B 0.000, C 0.000 }
gfCNCPoint6[1188] = {X 358.2611, Y 2.3048, Z -8.0000, A 0.000, B 0.000, C 0.000 }
gfCNCPoint6[1189] = {X 360.1227, Y 3.4745, Z -8.0000, A 0.000, B 0.000, C 0.000 }
gfCNCPoint6[1190] = {X 361.8557, Y 4.8274, Z -8.0000, A 0.000, B 0.000, C 0.000 }
gfCNCPoint6[1191] = {X 363.4420, Y 6.3496, Z -8.0000, A 0.000, B 0.000, C 0.000 }
gfCNCPoint6[1192] = {X 363.5023, Y 6.4139, Z -8.0000, A 0.000, B 0.000, C 0.000 }
gfCNCPoint6[1193] = {X 363.5623, Y 6.4785, Z -8.0000, A 0.000, B 0.000, C 0.000 }
gfCNCPoint6[1194] = {X 364.8945, Y 8.0610, Z -8.0000, A 0.000, B 0.000, C 0.000 }
gfCNCPoint6[1195] = {X 366.0933, Y 9.7469, Z -8.0000, A 0.000, B 0.000, C 0.000 }
gfCNCPoint6[1196] = {X 367.1506, Y 11.5249, Z -8.0000, A 0.000, B 0.000, C 0.000 }
gfCNCPoint6[1197] = {X 368.0594, Y 13.3832, Z -8.0000, A 0.000, B 0.000, C 0.000 }
gfCNCPoint6[1198] = {X 368.8137, Y 15.3095, Z -8.0000, A 0.000, B 0.000, C 0.000 }
gfCNCPoint6[1199] = {X 369.4084, Y 17.2908, Z -8.0000, A 0.000, B 0.000, C 0.000 }
gfCNCPoint6[1200] = {X 369.8996, Y 19.6246, Z -8.0000, A 0.000, B 0.000, C 0.000 }
gfCNCPoint6[1201] = {X 370.2164, Y 21.9885, Z -8.0000, A 0.000, B 0.000, C 0.000 }
gfCNCPoint6[1202] = {X 370.3570, Y 24.3694, Z -8.0000, A 0.000, B 0.000, C 0.000 }
gfCNCPoint6[1203] = {X 370.3207, Y 26.7541, Z -8.0000, A 0.000, B 0.000, C 0.000 }
gfCNCPoint6[1204] = {X 370.1077, Y 29.1295, Z -8.0000, A 0.000, B 0.000, C 0.000 }
gfCNCPoint6[1205] = {X 369.7191, Y 31.4827, Z -8.0000, A 0.000, B 0.000, C 0.000 }
gfCNCPoint6[1206] = {X 369.1832, Y 33.6343, Z -8.0000, A 0.000, B 0.000, C 0.000 }
gfCNCPoint6[1207] = {X 368.4594, Y 35.7303, Z -8.0000, A 0.000, B 0.000, C 0.000 }
gfCNCPoint6[1208] = {X 367.5534, Y 37.7542, Z -8.0000, A 0.000, B 0.000, C 0.000 }
gfCNCPoint6[1209] = {X 366.4724, Y 39.6902, Z -8.0000, A 0.000, B 0.000, C 0.000 }
gfCNCPoint6[1210] = {X 365.2247, Y 41.5232, Z -8.0000, A 0.000, B 0.000, C 0.000 }
gfCNCPoint6[1211] = {X 365.1111, Y 41.6784, Z -8.0000, A 0.000, B 0.000, C 0.000 }
gfCNCPoint6[1212] = {X 363.6765, Y 43.3979, Z -8.0000, A 0.000, B 0.000, C 0.000 }
gfCNCPoint6[1213] = {X 362.0784, Y 44.9667, Z -8.0000, A 0.000, B 0.000, C 0.000 }
gfCNCPoint6[1214] = {X 360.3326, Y 46.3691, Z -8.0000, A 0.000, B 0.000, C 0.000 }
gfCNCPoint6[1215] = {X 358.4562, Y 47.5915, Z -8.0000, A 0.000, B 0.000, C 0.000 }
gfCNCPoint6[1216] = {X 356.4678, Y 48.6216, Z -8.0000, A 0.000, B 0.000, C 0.000 }
gfCNCPoint6[1217] = {X 354.6708, Y 49.3155, Z -8.0000, A 0.000, B 0.000, C 0.000 }
gfCNCPoint6[1218] = {X 352.8231, Y 49.8605, Z -8.0000, A 0.000, B 0.000, C 0.000 }
gfCNCPoint6[1219] = {X 350.9372, Y 50.2528, Z -8.0000, A 0.000, B 0.000, C 0.000 }
gfCNCPoint6[1220] = {X 349.0255, Y 50.4899, Z -8.0000, A 0.000, B 0.000, C 0.000 }
gfCNCPoint6[1221] = {X 347.1008, Y 50.5702, Z -8.0000, A 0.000, B 0.000, C 0.000 }
gfCNCPoint6[1222] = {X 344.9874, Y 50.5340, Z -8.0000, A 0.000, B 0.000, C 0.000 }
gfCNCPoint6[1223] = {X 342.8851, Y 50.3148, Z -8.0000, A 0.000, B 0.000, C 0.000 }
gfCNCPoint6[1224] = {X 340.8096, Y 49.9142, Z -8.0000, A 0.000, B 0.000, C 0.000 }
